	(*Tooling position to load parts*)
	Tool_At_Load.0:=
				(((Model_ID=1) OR (Model_ID>3))		(*Model 504, 526, 536, 550, 571*)
				AND Clamp1RETD AND Clamp2RETD AND Clamp3RETD AND Clamp4RETD
				AND Clamp5RETD AND Clamp6RETD AND Clamp7RETD AND Clamp8RETD
				AND Clamp9RETD AND Clamp10RETD AND Clamp11RETD AND Clamp12RETD
				AND Clamp13RETD AND Clamp14RETD AND Clamp15RETD AND Clamp16RETD
				AND Clamp17RETD AND Clamp18RETD AND Clamp19RETD AND Clamp20RETD
				AND Clamp21RETD AND Clamp22RETD AND Pin1ADVD AND Pin2ADVD AND Pin3ADVD AND Pin4ADVD 
				AND Pin5RETD AND Pin6RETD AND Pin7ADVD AND Pin8ADVD AND Pin9ADVD AND Pin10ADVD 
				AND Pin11ADVD AND Pin12ADVD AND Pin13ADVD AND Pin14RETD AND Pin15RETD AND Pin16ADVD AND Pin17ADVD 
				AND Pin18ADVD AND Slide1ADVD AND Slide2ADVD AND Slide3RETD AND Slide4RETD AND Slide5RETD AND Slide6RETD
				AND Slide7RETD AND Slide8RETD AND Slide9RETD AND Slide10ADVD AND Slide11RETD AND Slide12RETD
				AND Slide13ADVD AND Slide14ADVD AND Swing1RETD AND Swing2RETD AND Swing3RETD)
			OR
				((Model_ID=2)		(*Model 524*)
				AND Clamp1RETD AND Clamp2RETD AND Clamp3RETD AND Clamp4RETD
				AND Clamp5RETD AND Clamp6RETD AND Clamp7RETD AND Clamp8RETD
				AND Clamp9RETD AND Clamp10RETD AND Clamp11RETD AND Clamp12RETD
				AND Clamp13RETD AND Clamp14RETD AND Clamp15RETD AND Clamp16RETD
				AND Clamp17RETD AND Clamp18RETD AND Clamp19RETD AND Clamp20RETD
				AND Clamp21RETD AND Clamp22RETD AND Pin1ADVD AND Pin2ADVD AND Pin3ADVD AND Pin4ADVD 
				AND Pin5ADVD AND Pin6RETD AND Pin7ADVD AND Pin8ADVD AND Pin9ADVD AND Pin10ADVD 
				AND Pin11ADVD AND Pin12ADVD AND Pin13ADVD AND Pin14RETD AND Pin15ADVD AND Pin16ADVD AND Pin17ADVD 
				AND Pin18ADVD AND Slide1ADVD AND Slide2ADVD AND Slide3RETD AND Slide4RETD AND Slide5RETD AND Slide6RETD
				AND Slide7RETD AND Slide8RETD AND Slide9RETD AND Slide10ADVD AND Slide11RETD AND Slide12RETD
				AND Slide13ADVD AND Slide14ADVD AND Swing1RETD AND Swing2RETD AND Swing3RETD)
			OR
				((Model_ID=3)		(*Model 543*)
				AND Clamp1RETD AND Clamp2RETD AND Clamp3RETD AND Clamp4RETD
				AND Clamp5RETD AND Clamp6RETD AND Clamp7RETD AND Clamp8RETD
				AND Clamp9RETD AND Clamp10RETD AND Clamp11RETD AND Clamp12RETD
				AND Clamp13RETD AND Clamp14RETD AND Clamp15RETD AND Clamp16RETD
				AND Clamp17RETD AND Clamp18RETD AND Clamp19RETD AND Clamp20RETD
				AND Clamp21RETD AND Clamp22RETD AND Pin1ADVD AND Pin2ADVD AND Pin3ADVD AND Pin4ADVD 
				AND Pin5RETD AND Pin6ADVD AND Pin7ADVD AND Pin8ADVD AND Pin9ADVD AND Pin10ADVD 
				AND Pin11ADVD AND Pin12ADVD AND Pin13ADVD AND Pin14ADVD AND Pin15RETD AND Pin16ADVD AND Pin17ADVD 
				AND Pin18ADVD AND Slide1ADVD AND Slide2ADVD AND Slide3RETD AND Slide4RETD AND Slide5RETD AND Slide6RETD
				AND Slide7RETD AND Slide8RETD AND Slide9RETD AND Slide10ADVD AND Slide11RETD AND Slide12RETD
				AND Slide13ADVD AND Slide14ADVD AND Swing1RETD AND Swing2RETD AND Swing3RETD);
	
	(*Tooling position on Loading Complete*)	
	Tool_At_Load.1:= 
				(((Model_ID=1) OR (Model_ID>3))		(*Model 504, 526, 536, 550, 571*)
				AND Clamp1ADVD AND Clamp2ADVD AND Clamp3ADVD AND Clamp4ADVD AND Clamp5ADVD AND Clamp5ADVD AND Clamp5ADVD
				AND Clamp6ADVD AND Clamp7ADVD AND Clamp8ADVD AND Clamp9ADVD AND Clamp10ADVD AND Clamp11ADVD AND Clamp12ADVD
				AND Clamp13ADVD AND Clamp14ADVD AND Clamp15ADVD AND Clamp16ADVD AND Clamp17ADVD AND Clamp18ADVD AND Clamp19ADVD
				AND Clamp20ADVD AND Clamp21ADVD AND Clamp22ADVD AND Pin1ADVD AND Pin2ADVD AND Pin3ADVD AND Pin4ADVD AND Pin5RETD
				AND Pin6RETD AND Pin7ADVD AND Pin8ADVD AND Pin9ADVD AND Pin10ADVD AND Pin11ADVD AND Pin12ADVD AND Pin13ADVD
				AND Pin14RETD AND Pin15RETD AND Pin16ADVD AND Pin17ADVD AND Pin18ADVD AND Slide1ADVD AND Slide2ADVD AND Slide3ADVD
				AND Slide4ADVD AND Slide5ADVD AND Slide6ADVD AND Slide7ADVD AND Slide8ADVD AND Slide9ADVD AND Slide10ADVD AND Slide11ADVD
				AND Slide12ADVD AND Slide13ADVD AND Slide14ADVD AND Swing1ADVD AND Swing2ADVD AND Swing3ADVD)
			OR
				((Model_ID=2)		(*Model 524*)
				AND Clamp1ADVD AND Clamp2ADVD AND Clamp3ADVD AND Clamp4ADVD AND Clamp5ADVD AND Clamp5ADVD AND Clamp5ADVD
				AND Clamp6ADVD AND Clamp7ADVD AND Clamp8ADVD AND Clamp9ADVD AND Clamp10ADVD AND Clamp11ADVD AND Clamp12ADVD
				AND Clamp13ADVD AND Clamp14ADVD AND Clamp15ADVD AND Clamp16ADVD AND Clamp17ADVD AND Clamp18ADVD AND Clamp19ADVD
				AND Clamp20ADVD AND Clamp21ADVD AND Clamp22ADVD AND Pin1ADVD AND Pin2ADVD AND Pin3ADVD AND Pin4ADVD AND Pin5ADVD
				AND Pin6RETD AND Pin7ADVD AND Pin8ADVD AND Pin9ADVD AND Pin10ADVD AND Pin11ADVD AND Pin12ADVD AND Pin13ADVD
				AND Pin14RETD AND Pin15ADVD AND Pin16ADVD AND Pin17ADVD AND Pin18ADVD AND Slide1ADVD AND Slide2ADVD AND Slide3ADVD
				AND Slide4ADVD AND Slide5ADVD AND Slide6ADVD AND Slide7ADVD AND Slide8ADVD AND Slide9ADVD AND Slide10ADVD AND Slide11ADVD
				AND Slide12ADVD AND Slide13ADVD AND Slide14ADVD AND Swing1ADVD AND Swing2ADVD AND Swing3ADVD)
			OR
				((Model_ID=3)		(*Model 543*)
				AND Clamp1ADVD AND Clamp2ADVD AND Clamp3ADVD AND Clamp4ADVD AND Clamp5ADVD AND Clamp5ADVD AND Clamp5ADVD
				AND Clamp6ADVD AND Clamp7ADVD AND Clamp8ADVD AND Clamp9ADVD AND Clamp10ADVD AND Clamp11ADVD AND Clamp12ADVD
				AND Clamp13ADVD AND Clamp14ADVD AND Clamp15ADVD AND Clamp16ADVD AND Clamp17ADVD AND Clamp18ADVD AND Clamp19ADVD
				AND Clamp20ADVD AND Clamp21ADVD AND Clamp22ADVD AND Pin1ADVD AND Pin2ADVD AND Pin3ADVD AND Pin4ADVD AND Pin5RETD
				AND Pin6ADVD AND Pin7ADVD AND Pin8ADVD AND Pin9ADVD AND Pin10ADVD AND Pin11ADVD AND Pin12ADVD AND Pin13ADVD
				AND Pin14ADVD AND Pin15RETD AND Pin16ADVD AND Pin17ADVD AND Pin18ADVD AND Slide1ADVD AND Slide2ADVD AND Slide3ADVD
				AND Slide4ADVD AND Slide5ADVD AND Slide6ADVD AND Slide7ADVD AND Slide8ADVD AND Slide9ADVD AND Slide10ADVD AND Slide11ADVD
				AND Slide12ADVD AND Slide13ADVD AND Slide14ADVD AND Swing1ADVD AND Swing2ADVD AND Swing3ADVD);
	(*Tool Position for Calling in Load Robots*)
	Tool_At_Load.2:=  
				(((Model_ID=1) OR (Model_ID>3))		(*Model 504, 526, 536, 550, 571*)
				AND Clamp1ADVD AND Clamp2ADVD AND Clamp3ADVD AND Clamp4ADVD AND Clamp5ADVD
				AND Clamp6RETD AND Clamp7RETD AND Clamp8RETD AND Clamp9ADVD AND Clamp10ADVD AND Clamp11RETD AND Clamp12ADVD
				AND Clamp13ADVD AND Clamp14ADVD AND Clamp15RETD AND Clamp16ADVD AND Clamp17RETD AND Clamp18ADVD AND Clamp19RETD
				AND Clamp20RETD AND Clamp21ADVD AND Clamp22ADVD AND Pin1ADVD AND Pin2ADVD AND Pin3ADVD AND Pin4ADVD AND Pin5RETD
				AND Pin6RETD AND Pin7ADVD AND Pin8ADVD AND Pin9ADVD AND Pin10ADVD AND Pin11ADVD AND Pin12ADVD AND Pin13ADVD
				AND Pin14RETD AND Pin15RETD AND Pin16ADVD AND Pin17ADVD AND Pin18ADVD AND Slide1ADVD AND Slide2ADVD AND Slide3RETD
				AND Slide4RETD AND Slide5RETD AND Slide6RETD AND Slide7RETD AND Slide8RETD AND Slide9RETD AND Slide10ADVD AND Slide11RETD
				AND Slide12RETD AND Slide13ADVD AND Slide14ADVD AND Swing1RETD AND Swing2RETD AND Swing3RETD)
			OR
				((Model_ID=2)		(*Model 524*)
				AND Clamp1ADVD AND Clamp2ADVD AND Clamp3ADVD AND Clamp4ADVD AND Clamp5ADVD
				AND Clamp6ADVD AND Clamp7RETD AND Clamp8RETD AND Clamp9ADVD AND Clamp10ADVD AND Clamp11RETD AND Clamp12ADVD
				AND Clamp13ADVD AND Clamp14ADVD AND Clamp15RETD AND Clamp16ADVD AND Clamp17RETD AND Clamp18ADVD AND Clamp19RETD
				AND Clamp20ADVD AND Clamp21ADVD AND Clamp22ADVD AND Pin1ADVD AND Pin2ADVD AND Pin3ADVD AND Pin4ADVD AND Pin5ADVD
				AND Pin6RETD AND Pin7ADVD AND Pin8ADVD AND Pin9ADVD AND Pin10ADVD AND Pin11ADVD AND Pin12ADVD AND Pin13ADVD
				AND Pin14RETD AND Pin15ADVD AND Pin16ADVD AND Pin17ADVD AND Pin18ADVD AND Slide1ADVD AND Slide2ADVD AND Slide3RETD
				AND Slide4RETD AND Slide5RETD AND Slide6RETD AND Slide7RETD AND Slide8RETD AND Slide9RETD AND Slide10ADVD AND Slide11RETD
				AND Slide12RETD AND Slide13ADVD AND Slide14ADVD AND Swing1RETD AND Swing2RETD AND Swing3RETD)
			OR
				((Model_ID=3)		(*Model 543*)
				AND Clamp1ADVD AND Clamp2ADVD AND Clamp3ADVD AND Clamp4ADVD AND Clamp5ADVD
				AND Clamp6RETD AND Clamp7RETD AND Clamp8ADVD AND Clamp9ADVD AND Clamp10ADVD AND Clamp11RETD AND Clamp12ADVD
				AND Clamp13ADVD AND Clamp14ADVD AND Clamp15RETD AND Clamp16ADVD AND Clamp17RETD AND Clamp18ADVD AND Clamp19ADVD
				AND Clamp20RETD AND Clamp21ADVD AND Clamp22ADVD AND Pin1ADVD AND Pin2ADVD AND Pin3ADVD AND Pin4ADVD AND Pin5RETD
				AND Pin6ADVD AND Pin7ADVD AND Pin8ADVD AND Pin9ADVD AND Pin10ADVD AND Pin11ADVD AND Pin12ADVD AND Pin13ADVD
				AND Pin14ADVD AND Pin15RETD AND Pin16ADVD AND Pin17ADVD AND Pin18ADVD AND Slide1ADVD AND Slide2ADVD AND Slide3RETD
				AND Slide4RETD AND Slide5RETD AND Slide6RETD AND Slide7RETD AND Slide8RETD AND Slide9RETD AND Slide10ADVD AND Slide11RETD
				AND Slide12RETD AND Slide13ADVD AND Slide14ADVD AND Swing1RETD AND Swing2RETD AND Swing3RETD);
	Tool_At_Load.3:= FALSE;
	Tool_At_Load.4:= FALSE;


	Tool_At_Seal.0:= FALSE;
	Tool_At_Seal.1:= FALSE;
	Tool_At_Seal.2:= FALSE;
	Tool_At_Seal.3:= FALSE;
	Tool_At_Seal.4:= FALSE;


	Tool_At_Stud.0:= FALSE;
	Tool_At_Stud.1:= FALSE;
	Tool_At_Stud.2:= FALSE;
	Tool_At_Stud.3:= FALSE;
	Tool_At_Stud.4:= FALSE;

	(*Tooling position for ready to rotate*)
	Tool_At_Rotate.0:= 
				(((Model_ID=1) OR (Model_ID>3))		(*Model 504, 526, 536, 550, 571*)
				AND Clamp1ADVD AND Clamp2ADVD AND Clamp3ADVD AND Clamp4ADVD AND Clamp5ADVD
				AND Clamp6RETD AND Clamp7RETD AND Clamp8RETD AND Clamp9ADVD AND Clamp10ADVD AND Clamp11RETD AND Clamp12ADVD
				AND Clamp13ADVD AND Clamp14ADVD AND Clamp15RETD AND Clamp16ADVD AND Clamp17RETD AND Clamp18ADVD AND Clamp19RETD
				AND Clamp20RETD AND Clamp21ADVD AND Clamp22ADVD AND Pin1ADVD AND Pin2ADVD AND Pin3ADVD AND Pin4ADVD AND Pin5RETD
				AND Pin6RETD AND Pin7ADVD AND Pin8ADVD AND Pin9ADVD AND Pin10ADVD AND Pin11ADVD AND Pin12ADVD AND Pin13ADVD
				AND Pin14RETD AND Pin15RETD AND Pin16ADVD AND Pin17ADVD AND Pin18ADVD AND Slide1ADVD AND Slide2ADVD AND Slide3RETD
				AND Slide4RETD AND Slide5RETD AND Slide6RETD AND Slide7RETD AND Slide8RETD AND Slide9RETD AND Slide10ADVD AND Slide11RETD
				AND Slide12RETD AND Slide13ADVD AND Slide14ADVD AND Swing1RETD AND Swing2RETD AND Swing3RETD)
			OR
				((Model_ID=2)		(*Model 524*)
				AND Clamp1ADVD AND Clamp2ADVD AND Clamp3ADVD AND Clamp4ADVD AND Clamp5ADVD
				AND Clamp6ADVD AND Clamp7RETD AND Clamp8RETD AND Clamp9ADVD AND Clamp10ADVD AND Clamp11RETD AND Clamp12ADVD
				AND Clamp13ADVD AND Clamp14ADVD AND Clamp15RETD AND Clamp16ADVD AND Clamp17RETD AND Clamp18ADVD AND Clamp19RETD
				AND Clamp20ADVD AND Clamp21ADVD AND Clamp22ADVD AND Pin1ADVD AND Pin2ADVD AND Pin3ADVD AND Pin4ADVD AND Pin5ADVD
				AND Pin6RETD AND Pin7ADVD AND Pin8ADVD AND Pin9ADVD AND Pin10ADVD AND Pin11ADVD AND Pin12ADVD AND Pin13ADVD
				AND Pin14RETD AND Pin15ADVD AND Pin16ADVD AND Pin17ADVD AND Pin18ADVD AND Slide1ADVD AND Slide2ADVD AND Slide3RETD
				AND Slide4RETD AND Slide5RETD AND Slide6RETD AND Slide7RETD AND Slide8RETD AND Slide9RETD AND Slide10ADVD AND Slide11RETD
				AND Slide12RETD AND Slide13ADVD AND Slide14ADVD AND Swing1RETD AND Swing2RETD AND Swing3RETD)
			OR
				((Model_ID=3)		(*Model 543*)
				AND Clamp1ADVD AND Clamp2ADVD AND Clamp3ADVD AND Clamp4ADVD AND Clamp5ADVD
				AND Clamp6RETD AND Clamp7RETD AND Clamp8ADVD AND Clamp9ADVD AND Clamp10ADVD AND Clamp11RETD AND Clamp12ADVD
				AND Clamp13ADVD AND Clamp14ADVD AND Clamp15RETD AND Clamp16ADVD AND Clamp17RETD AND Clamp18ADVD AND Clamp19ADVD
				AND Clamp20RETD AND Clamp21ADVD AND Clamp22ADVD AND Pin1ADVD AND Pin2ADVD AND Pin3ADVD AND Pin4ADVD AND Pin5RETD
				AND Pin6ADVD AND Pin7ADVD AND Pin8ADVD AND Pin9ADVD AND Pin10ADVD AND Pin11ADVD AND Pin12ADVD AND Pin13ADVD
				AND Pin14ADVD AND Pin15RETD AND Pin16ADVD AND Pin17ADVD AND Pin18ADVD AND Slide1ADVD AND Slide2ADVD AND Slide3RETD
				AND Slide4RETD AND Slide5RETD AND Slide6RETD AND Slide7RETD AND Slide8RETD AND Slide9RETD AND Slide10ADVD AND Slide11RETD
				AND Slide12RETD AND Slide13ADVD AND Slide14ADVD AND Swing1RETD AND Swing2RETD AND Swing3RETD);
				
	Tool_At_Rotate.1:= FALSE;
	Tool_At_Rotate.2:= FALSE;
	Tool_At_Rotate.3:= FALSE;
	Tool_At_Rotate.4:= FALSE;

	(*Tooling position for welding*)
	Tool_At_Weld.0:= 
				(((Model_ID=1) OR (Model_ID>3))		(*Model 504, 526, 536, 550, 571*)
				AND Clamp1ADVD AND Clamp2ADVD AND Clamp3ADVD AND Clamp4ADVD AND Clamp5ADVD AND Clamp5ADVD AND Clamp5ADVD
				AND Clamp6RETD AND Clamp7ADVD AND Clamp8RETD AND Clamp9ADVD AND Clamp10ADVD AND Clamp11ADVD AND Clamp12ADVD
				AND Clamp13ADVD AND Clamp14ADVD AND Clamp15ADVD AND Clamp16ADVD AND Clamp17ADVD AND Clamp18ADVD AND Clamp19RETD
				AND Clamp20RETD AND Clamp21ADVD AND Clamp22ADVD AND Pin1ADVD AND Pin2ADVD AND Pin3ADVD AND Pin4ADVD AND Pin5RETD
				AND Pin6RETD AND Pin7ADVD AND Pin8ADVD AND Pin9ADVD AND Pin10ADVD AND Pin11ADVD AND Pin12ADVD AND Pin13ADVD
				AND Pin14RETD AND Pin15RETD AND Pin16ADVD AND Pin17ADVD AND Pin18ADVD AND Slide1ADVD AND Slide2ADVD AND Slide3ADVD
				AND Slide4RETD AND Slide5ADVD AND Slide6ADVD AND Slide7ADVD AND Slide8ADVD AND Slide9ADVD AND Slide10ADVD AND Slide11RETD
				AND Slide12ADVD AND Slide13ADVD AND Slide14ADVD AND Swing1RETD AND Swing2ADVD AND Swing3RETD)
			OR
				((Model_ID=2)		(*Model 524*)
				AND Clamp1ADVD AND Clamp2ADVD AND Clamp3ADVD AND Clamp4ADVD AND Clamp5ADVD AND Clamp5ADVD AND Clamp5ADVD
				AND Clamp6ADVD AND Clamp7ADVD AND Clamp8RETD AND Clamp9ADVD AND Clamp10ADVD AND Clamp11ADVD AND Clamp12ADVD
				AND Clamp13ADVD AND Clamp14ADVD AND Clamp15ADVD AND Clamp16ADVD AND Clamp17ADVD AND Clamp18ADVD AND Clamp19RETD
				AND Clamp20ADVD AND Clamp21ADVD AND Clamp22ADVD AND Pin1ADVD AND Pin2ADVD AND Pin3ADVD AND Pin4ADVD AND Pin5ADVD
				AND Pin6RETD AND Pin7ADVD AND Pin8ADVD AND Pin9ADVD AND Pin10ADVD AND Pin11ADVD AND Pin12ADVD AND Pin13ADVD
				AND Pin14RETD AND Pin15ADVD AND Pin16ADVD AND Pin17ADVD AND Pin18ADVD AND Slide1ADVD AND Slide2ADVD AND Slide3ADVD
				AND Slide4ADVD AND Slide5ADVD AND Slide6ADVD AND Slide7ADVD AND Slide8ADVD AND Slide9ADVD AND Slide10ADVD AND Slide11ADVD
				AND Slide12ADVD AND Slide13ADVD AND Slide14ADVD AND Swing1RETD AND Swing2ADVD AND Swing3RETD)
			OR
				((Model_ID=3)		(*Model 543*)
				AND Clamp1ADVD AND Clamp2ADVD AND Clamp3ADVD AND Clamp4ADVD AND Clamp5ADVD AND Clamp5ADVD AND Clamp5ADVD
				AND Clamp6RETD AND Clamp7ADVD AND Clamp8ADVD AND Clamp9ADVD AND Clamp10ADVD AND Clamp11ADVD AND Clamp12ADVD
				AND Clamp13ADVD AND Clamp14ADVD AND Clamp15ADVD AND Clamp16ADVD AND Clamp17ADVD AND Clamp18ADVD AND Clamp19ADVD
				AND Clamp20RETD AND Clamp21ADVD AND Clamp22ADVD AND Pin1ADVD AND Pin2ADVD AND Pin3ADVD AND Pin4ADVD AND Pin5RETD
				AND Pin6ADVD AND Pin7ADVD AND Pin8ADVD AND Pin9ADVD AND Pin10ADVD AND Pin11ADVD AND Pin12ADVD AND Pin13ADVD
				AND Pin14ADVD AND Pin15RETD AND Pin16ADVD AND Pin17ADVD AND Pin18ADVD AND Slide1ADVD AND Slide2ADVD AND Slide3ADVD
				AND Slide4RETD AND Slide5ADVD AND Slide6ADVD AND Slide7ADVD AND Slide8ADVD AND Slide9ADVD AND Slide10ADVD AND Slide11RETD
				AND Slide12ADVD AND Slide13ADVD AND Slide14ADVD AND Swing1ADVD AND Swing2ADVD AND Swing3ADVD);
	Tool_At_Weld.1:= FALSE;
	Tool_At_Weld.2:= FALSE;
	Tool_At_Weld.3:= FALSE;
	Tool_At_Weld.4:= FALSE;

	(*Tooling position for unload*)
	Tool_At_Unload.0:=Clamp1RETD AND Clamp2RETD AND Clamp3RETD AND Clamp4RETD
				AND Clamp5RETD AND Clamp6RETD AND Clamp7ADVD AND Clamp8RETD
				AND Clamp9RETD AND Clamp10RETD AND Clamp11ADVD AND Clamp12RETD
				AND Clamp13RETD AND Clamp14RETD AND Clamp15ADVD AND Clamp16RETD
				AND Clamp17ADVD AND Clamp18RETD AND Clamp19RETD AND Clamp20RETD
				AND Clamp21RETD AND Clamp22RETD AND Pin1RETD AND Pin2RETD AND Pin3RETD AND Pin4RETD AND Pin5RETD
				AND Pin6RETD AND Pin7RETD AND Pin8RETD AND Pin9RETD AND Pin10RETD AND Pin11RETD AND Pin12RETD 
				AND Pin13RETD AND Pin14RETD AND Pin15RETD AND Pin16RETD AND Pin17RETD AND Pin18RETD
				AND Slide1RETD AND Slide2RETD AND Slide3RETD AND Slide4RETD AND Slide5RETD AND Slide6RETD
				AND Slide7RETD AND Slide8RETD AND Slide9RETD AND Slide10RETD AND Slide11RETD AND Slide12RETD
				AND Slide13RETD AND Slide14RETD AND Swing1RETD AND Swing2RETD AND Swing3RETD;
	
	Tool_At_Unload.1:=Clamp1RETD AND Clamp2RETD AND Clamp3RETD AND Clamp4RETD
				AND Clamp5RETD AND Clamp6RETD AND Clamp7RETD AND Clamp8RETD
				AND Clamp9RETD AND Clamp10RETD AND Clamp11RETD AND Clamp12RETD
				AND Clamp13RETD AND Clamp14RETD AND Clamp15RETD AND Clamp16RETD
				AND Clamp17RETD AND Clamp18RETD AND Clamp19RETD AND Clamp20RETD
				AND Clamp21RETD AND Clamp22RETD AND Pin1RETD AND Pin2RETD AND Pin3RETD AND Pin4RETD AND Pin5RETD
				AND Pin6RETD AND Pin7RETD AND Pin8RETD AND Pin9RETD AND Pin10RETD AND Pin11RETD AND Pin12RETD 
				AND Pin13RETD AND Pin14RETD AND Pin15RETD AND Pin16RETD AND Pin17RETD AND Pin18RETD
				AND Slide1RETD AND Slide2RETD AND Slide3RETD AND Slide4RETD AND Slide5RETD AND Slide6RETD
				AND Slide7RETD AND Slide8RETD AND Slide9RETD AND Slide10RETD AND Slide11RETD AND Slide12RETD
				AND Slide13RETD AND Slide14RETD AND Swing1RETD AND Swing2RETD AND Swing3RETD;
	Tool_At_Unload.2:= FALSE;
	Tool_At_Unload.3:= FALSE;
	Tool_At_Unload.4:= FALSE;







































(*end*)
END_ACTION

ACTION Tool_VBSeq_Repos:
(*+++++++++++THIS AREA IS CUSTOM PER INSTALLATION AND WILL HAVE TO BE MODIFIED PER +++++++++++++*)
(*+++++++++++THIS AREA IS CUSTOM PER INSTALLATION AND WILL HAVE TO BE MODIFIED PER +++++++++++++*)


(*!!!!!!!!!!!!!!!!!!!!!!!!!!!!!!!!!!!!!!!!!! Tool Motion Control !!!!!!!!!!!!!!!!!!!!!!!!!!!!!!!*)

(*----------------------------------------- Clamp / Unclamp Steps -------------------------------*)

(*$$$$$$$$$$$$$$$$$$$$$$$$$$$$$$$$$$ Develop Clamp and Unclamp Interlocks $$$$$$$$$$$$$$$$$$$$$$*)
(* Note: This is one method to create valve bank commands for clamp and unclamp sequencing
you are welcome to use the direct method as well*)


	(*---------------------------------------------------------Start Clamp Sequence---------------------------------------------------------*)
	
	(*First Stage Clamping*)		(*V8, V10 ADV, IF Model 2 then V2 ADV, IF Model 3 then V5 ADV*)
	Clamp_Step.0:= Auto_Run AND NOT Welding_Complete OR (Cycle_Complete AND NOT Tool_At_Home AND All_Sensors_Off);
	
	
	(*Second Stage Clamping*)		(*V7, V9, V11 ADV, IF Model 2 then V1 ADV, IF Model 3 V4 ADV*)
	
	(*Model 504, 526, 536, 550, 571*)
	IF (Model_ID=1) OR (Model_ID>3) THEN		
				Clamp_Step.1:=  Clamp_Step.0 AND (Load_Complete1 OR Load_Complete2) AND
								(*V8*)
								(Pin1ADVD AND Pin2ADVD AND Pin3ADVD AND Pin4ADVD AND Pin7ADVD 
								AND Pin9ADVD AND Pin16ADVD AND Pin17ADVD AND Pin18ADVD AND Slide10ADVD)
								(*V10*)
								AND (Pin8ADVD AND Pin10ADVD AND Pin11ADVD AND Pin12ADVD AND Pin13ADVD 
								AND Slide1ADVD AND Slide2ADVD AND Slide13ADVD AND Slide14ADVD);
		(*Model 524*)						
		ELSIF (Model_ID=2) THEN					
				Clamp_Step.1:=  Clamp_Step.0 AND (Load_Complete1 OR Load_Complete2) AND
								(*V2*)
								(Pin5ADVD AND Pin15ADVD)
								(*V8*)
								AND (Pin1ADVD AND Pin2ADVD AND Pin3ADVD AND Pin4ADVD AND Pin7ADVD 
								AND Pin9ADVD AND Pin16ADVD AND Pin17ADVD AND Pin18ADVD AND Slide10ADVD)
								(*V10*)
								AND (Pin8ADVD AND Pin10ADVD AND Pin11ADVD AND Pin12ADVD AND Pin13ADVD 
								AND Slide1ADVD AND Slide2ADVD AND Slide13ADVD AND Slide14ADVD);
		(*Model 543*)			
		ELSIF (Model_ID=3) THEN					
				Clamp_Step.1:=  Clamp_Step.0 AND (Load_Complete1 OR Load_Complete2) AND 
								(*V5*)
								(Pin6ADVD AND Pin14ADVD)
								(*V8*)
								AND (Pin1ADVD AND Pin2ADVD AND Pin3ADVD AND Pin4ADVD AND Pin7ADVD 
								AND Pin9ADVD AND Pin16ADVD AND Pin17ADVD AND Pin18ADVD AND Slide10ADVD)
								(*V10*)
								AND (Pin8ADVD AND Pin10ADVD AND Pin11ADVD AND Pin12ADVD AND Pin13ADVD 
								AND Slide1ADVD AND Slide2ADVD AND Slide13ADVD AND Slide14ADVD);						
	END_IF

	
	(*Third Stage Clamping*)		(*V13 ADV*)
	
	(*Model 504, 526, 536, 550, 571*)
	IF (Model_ID=1) OR (Model_ID>3) THEN
				Clamp_Step.2:= 	Clamp_Step.1 AND (All_Sensors_On.2 OR Clamp_Step.2) AND Repo_Reqs.0 AND
								(*V7*)
								(Clamp3ADVD AND Clamp18ADVD)
								(*V9*)
								AND (Clamp1ADVD AND Clamp2ADVD AND Clamp4ADVD AND Clamp5ADVD AND Clamp10ADVD 
								AND Clamp14ADVD AND Clamp21ADVD AND Clamp22ADVD)
								(*V11*)
								AND (Clamp9ADVD AND Clamp12ADVD AND Clamp13ADVD AND Clamp16ADVD);

		ELSIF (Model_ID=2) THEN
				Clamp_Step.2:= 	Clamp_Step.1 AND (All_Sensors_On.2 OR Clamp_Step.2) AND Repo_Reqs.0 AND
								(*V7*)
								(Clamp3ADVD AND Clamp18ADVD)
								(*V9*)
								AND (Clamp1ADVD AND Clamp2ADVD AND Clamp4ADVD AND Clamp5ADVD AND Clamp10ADVD 
								AND Clamp14ADVD AND Clamp21ADVD AND Clamp22ADVD)
								(*V11*)
								AND (Clamp9ADVD AND Clamp12ADVD AND Clamp13ADVD AND Clamp16ADVD)
								(*V1*)
								AND (Clamp6ADVD AND Clamp20ADVD);
		ELSIF (Model_ID=3) THEN
				Clamp_Step.2:= 	Clamp_Step.1 AND (All_Sensors_On.2 OR Clamp_Step.2) AND Repo_Reqs.0 AND
								(*V7*)
								(Clamp3ADVD AND Clamp18ADVD)
								(*V9*)
								AND (Clamp1ADVD AND Clamp2ADVD AND Clamp4ADVD AND Clamp5ADVD AND Clamp10ADVD 
								AND Clamp14ADVD AND Clamp21ADVD AND Clamp22ADVD)
								(*V11*)
								AND (Clamp9ADVD AND Clamp12ADVD AND Clamp13ADVD AND Clamp16ADVD)
								(*V4*)
								AND (Clamp8ADVD AND Clamp19ADVD);
	END_IF


	(*Forth Stage Clamping*)		(*V12 ADV, IF Model 2 V3 ADV, IF Model 3 V6 ADV*)
	
	Clamp_Step.3:= Clamp_Step.2 AND Repo_Reqs.0 AND
					(*V13*)
					(Clamp7ADVD AND Clamp11ADVD AND Clamp15ADVD AND Clamp17ADVD);




	(*---------------------------------------------------------Start Unclamp Sequence---------------------------------------------------------*)

	(*First Stage Unclamping*)		(*V7, V9, V11 RET, IF Model 2 V1 RET, IF Model 3 V4 RET*)

	Unclamp_Step.0:= (Welding_Complete AND TurnTableA_At_Robot);


	(*Second Stage Unclamping*)		(*V8, V10 RET, IF Model 2 V2 RET, IF Model 3 V5 RET*)
	(*Model 504, 526, 536, 550, 571*)
	IF (Model_ID=1) OR (Model_ID>3) THEN
			Unclamp_Step.1:= Unclamp_Step.0 AND 
								(*V7*)
								(Clamp3RETD AND Clamp18RETD)
								(*V9*)
								AND (Clamp1RETD AND Clamp2RETD AND Clamp4RETD AND Clamp5RETD AND Clamp10RETD AND Clamp14RETD AND Clamp21RETD AND Clamp22RETD)
								(*V11*)
								AND (Clamp9RETD AND Clamp12RETD AND Clamp13RETD AND Clamp16RETD);
		(*Model 524*)							
		ELSIF (Model_ID=2) THEN
				Unclamp_Step.1:= Unclamp_Step.0 AND 
									(*V7*)
									(Clamp3RETD AND Clamp18RETD)
									(*V9*)
									AND (Clamp1RETD AND Clamp2RETD AND Clamp4RETD AND Clamp5RETD AND Clamp10RETD AND Clamp14RETD AND Clamp21RETD AND Clamp22RETD)
									(*V11*)
									AND (Clamp9RETD AND Clamp12RETD AND Clamp13RETD AND Clamp16RETD)
									(*V1*)
									AND (Clamp6RETD AND Clamp20RETD);
		(*Model 543*)
		ELSIF (Model_ID=3) THEN							
				Unclamp_Step.1:= Unclamp_Step.0 AND 
									(*V7*)
									(Clamp3RETD AND Clamp18RETD)
									(*V9*)
									AND (Clamp1RETD AND Clamp2RETD AND Clamp4RETD AND Clamp5RETD AND Clamp10RETD AND Clamp14RETD AND Clamp21RETD AND Clamp22RETD)
									(*V11*)
									AND (Clamp9RETD AND Clamp12RETD AND Clamp13RETD AND Clamp16RETD)
									(*V4*)
									AND (Clamp8RETD AND Clamp19RETD);
	END_IF

	
	(*Third Stage Unclamping*)		(*V12 RET, IF Model 2 V3 RET, IF Model 3 V6 RET*)
	(*Model 504, 526, 536, 550, 571*)
	IF (Model_ID=1) OR (Model_ID>3) THEN
			Unclamp_Step.2:= Unclamp_Step.1 AND 
						(*V8*)
						(Pin1RETD AND Pin2RETD AND Pin3RETD AND Pin4RETD AND Pin7RETD AND Pin9RETD AND Pin16RETD AND Pin17RETD AND Pin18RETD AND Slide10RETD)
						(*V10*)
						AND (Pin8RETD AND Pin10RETD AND Pin11RETD AND Pin12RETD AND Pin13RETD AND Slide1RETD AND Slide2RETD AND Slide13RETD AND Slide14RETD);
		(*Model 524*)
		ELSIF (Model_ID=2) THEN
				Unclamp_Step.2:= Unclamp_Step.1 AND 
							(*V8*)
							(Pin1RETD AND Pin2RETD AND Pin3RETD AND Pin4RETD AND Pin7RETD AND Pin9RETD AND Pin16RETD AND Pin17RETD AND Pin18RETD AND Slide10RETD)
							(*V10*)
							AND (Pin8RETD AND Pin10RETD AND Pin11RETD AND Pin12RETD AND Pin13RETD AND Slide1RETD AND Slide2RETD AND Slide13RETD AND Slide14RETD)
							(*V2*)
							AND (Pin5RETD AND Pin15RETD);
		(*Model 543*)
		ELSIF (Model_ID=3) THEN
				Unclamp_Step.2:= Unclamp_Step.1 AND 
							(*V8*)
							(Pin1RETD AND Pin2RETD AND Pin3RETD AND Pin4RETD AND Pin7RETD AND Pin9RETD AND Pin16RETD AND Pin17RETD AND Pin18RETD AND Slide10RETD)
							(*V10*)
							AND (Pin8RETD AND Pin10RETD AND Pin11RETD AND Pin12RETD AND Pin13RETD AND Slide1RETD AND Slide2RETD AND Slide13RETD AND Slide14RETD)
							(*V5*)
							AND (Pin6RETD AND Pin14RETD);
	
	END_IF

	(*Fourth Stage Unclamping*)		(*V13 RET*)
	(*Model 504, 526, 536, 550, 571*)
	IF (Model_ID=1) OR (Model_ID>3) THEN
				Unclamp_Step.3:= Unclamp_Step.2 AND Repo_Reqs.1 AND
							(*V12*)
							(Slide3RETD AND Slide5RETD AND Slide6RETD AND Slide7RETD AND Slide8RETD AND Slide9RETD AND Slide12RETD AND Swing2RETD);

		ELSIF (Model_ID=2) THEN
				Unclamp_Step.3:= Unclamp_Step.2 AND Repo_Reqs.1 AND 
							(*V12*)
							(Slide3RETD AND Slide5RETD AND Slide6RETD AND Slide7RETD AND Slide8RETD AND Slide9RETD AND Slide12RETD AND Swing2RETD)
							(*V3*)
							AND (Slide4RETD AND Slide11RETD);
							
							
		ELSIF (Model_ID=3) THEN
				Unclamp_Step.3:= Unclamp_Step.2 AND Repo_Reqs.1 AND 
							(*V12*)
							(Slide3RETD AND Slide5RETD AND Slide6RETD AND Slide7RETD AND Slide8RETD AND Slide9RETD AND Slide12RETD AND Swing2RETD)
							(*V6*)
							AND (Swing1RETD AND Swing3RETD);
							
	END_IF							


(*------------------------------------------- Repositions --------------------------------------*)

	(*Reposition Request#1*)
	IF (MAIN.R4.Peripheral_Req.0 AND (MAIN.R4.Task_ID_Ack=DropOff_Fix03))
		THEN
			Repo_Reqs.0:= TRUE;
	END_IF;

	(*Reposition Request#2*)
	IF (MAIN.R4.Peripheral_Req.1 AND (MAIN.R4.Task_ID_Ack=Pickup_Fix03))
		THEN
			Repo_Reqs.1:= TRUE;
	END_IF;

	(*Reposition Request#3*)
	IF FALSE
		THEN
			Repo_Reqs.2:= TRUE;
	END_IF;

	(*Reposition Request#4*)
	IF FALSE
		THEN
			Repo_Reqs.3:= TRUE;
	END_IF;

	(*Reposition Request#5*)
	IF FALSE
		THEN
			Repo_Reqs.4:= TRUE;
	END_IF;

	(*Reposition Request#6*)
	IF FALSE
		THEN
			Repo_Reqs.5:= TRUE;
	END_IF;

	(*Reposition Request#7*)
	IF FALSE
		THEN
			Repo_Reqs.6:= TRUE;
	END_IF;

	(*Reposition Request#8*)
	IF FALSE
		THEN
			Repo_Reqs.7:= TRUE;
	END_IF;

	(*Reset All Reposition Acks At the End Of Cycle*)
	IF Cycle_Complete
		THEN
			Repo_Reqs:= 0;
	END_IF;

(*------------------------- Reposition Acks ---------------------*)
	Repo_Ack.0:= Repo_Reqs.0 AND All_Sensors_On.2 AND Tool_At_Weld.0;
	Repo_Ack.1:= Repo_Reqs.1 AND All_Sensors_On.8 AND Tool_At_Unload.1;
	Repo_Ack.2:= Repo_Reqs.2 AND FALSE;
	Repo_Ack.3:= Repo_Reqs.3 AND FALSE;
	Repo_Ack.4:= Repo_Reqs.4 AND FALSE;
	Repo_Ack.5:= Repo_Reqs.5 AND FALSE;
	Repo_Ack.6:= Repo_Reqs.6 AND FALSE;
	Repo_Ack.7:= Repo_Reqs.7 AND FALSE;
END_ACTION

ACTION ValveBank1:


(*+++++++++++THIS AREA IS CUSTOM PER INSTALLATION AND WILL HAVE TO BE MODIFIED PER +++++++++++++*)
(*+++++++++++THIS AREA IS CUSTOM PER INSTALLATION AND WILL HAVE TO BE MODIFIED PER +++++++++++++*)
(*+++++++++++THIS AREA IS CUSTOM PER INSTALLATION AND WILL HAVE TO BE MODIFIED PER +++++++++++++*)

(*+++++++++++VALVE BANK 1 +++++++++++++*)
(*+++++++++++VALVE BANK 1 +++++++++++++*)
(*+++++++++++VALVE BANK 1 +++++++++++++*)


	(*Valve 1, Model 524 ONLY*)
	(*Clamp #6, 20*)
		Valve1FB
			(
			Enable_Motion:= Enable_Motion,
			Enable_Latch:= TRUE,					(*Enabling Runs Valve as detent type (maintained solenoids*)
			Enable_SideA_PreCharge:= FALSE,		(*Enabling Turns Side A PreCharge Active, reset when Side B is energized in Auto*)
			Enable_SideB_PreCharge:= FALSE,		(*Enabling Turns Side B PreCharge Active, reset when Side A is energized in Auto*)
			PreCharge_Time:= T#0.1S,
			Enable_Auto_Commands:= In_Auto,
			Enable_Manual_Commands:= In_Manual AND (All_Robots_Clear OR TurntableB_At_Robot),  (*TLK ADDED OR*)
			In_Manual_SideA_Command:= Discrete_In.ManReqs.0,
			In_Manual_SideB_Command:= (Discrete_In.ManReqs.1 OR Discrete_In.Go_Home),
			SideA_Indicator:= (Clamp6ADVD AND Clamp20ADVD),
			SideB_Indicator:= (Clamp6RETD AND Clamp20RETD) OR Manual_Ind_HomePrompt,
			TurnOn_SideA_SOL=> N100.Q.0,
			TurnOn_SideB_SOL=> N100.Q.1,
			TurnOn_SideA_Indicator=> Manual_Indicators1.0,
			TurnOn_SideB_Indicator=> Manual_Indicators1.1
			 );
	IF (Model_ID=2) THEN		 
			Valve1FB.In_Auto_SideA_Command:= Clamp_Step.1 AND NOT Unclamp_Step.0;
			Valve1FB.In_Auto_SideB_Command:= Unclamp_Step.0 
										OR ((TurntableA_At_Robot OR Turntable_Bypassed) AND All_Sensors_Off AND Weld_Robots_Clear);
		ELSE
			Valve1FB.In_Auto_SideA_Command:= FALSE;
			Valve1FB.In_Auto_SideB_Command:= TRUE;
		END_IF

	(*Valve 2, Model 524 ONLY*)
	(*Pin #5, 15*)
		Valve2FB
			(
			Enable_Motion:= Enable_Motion,
			Enable_Latch:= TRUE,					(*Enabling Runs Valve as detent type (maintained solenoids*)
			Enable_SideA_PreCharge:= FALSE,		(*Enabling Turns Side A PreCharge Active, reset when Side B is energized in Auto*)
			Enable_SideB_PreCharge:= FALSE,		(*Enabling Turns Side B PreCharge Active, reset when Side A is energized in Auto*)
			PreCharge_Time:= T#0.10S,
			Enable_Auto_Commands:= In_Auto,
			Enable_Manual_Commands:= In_Manual AND (All_Robots_Clear OR TurntableB_At_Robot),  (*TLK ADDED OR*)
			In_Manual_SideA_Command:=  (Discrete_In.ManReqs.2 OR (Discrete_In.Go_Home AND (Model_ID = 2))),
			In_Manual_SideB_Command:= (Discrete_In.ManReqs.3 OR (Discrete_In.Go_Home AND (Model_ID <> 2))),
			SideA_Indicator:=  Pin5ADVD AND Pin15ADVD,
			SideB_Indicator:= (Pin5RETD AND Pin15RETD) OR Manual_Ind_HomePrompt,
			TurnOn_SideA_SOL=> N100.Q.2,
			TurnOn_SideB_SOL=> N100.Q.3,
			TurnOn_SideA_Indicator=> Manual_Indicators1.2,
			TurnOn_SideB_Indicator=> Manual_Indicators1.3
			 );
	IF (Model_ID=2) THEN		 
			Valve2FB.In_Auto_SideA_Command:= Clamp_Step.0 AND NOT Unclamp_Step.1
										OR ((TurntableA_At_Robot OR Turntable_Bypassed) AND All_Sensors_Off AND Weld_Robots_Clear);
			Valve2FB.In_Auto_SideB_Command:= Unclamp_Step.1;
		ELSE
			Valve2FB.In_Auto_SideA_Command:= FALSE;
			Valve2FB.In_Auto_SideB_Command:= TRUE;
		END_IF

	(*Valve 3, Model 524 ONLY*)
	(*Slide #4, 11*)
		Valve3FB
			(
			Enable_Motion:= Enable_Motion,
			Enable_Latch:= TRUE,					(*Enabling Runs Valve as detent type (maintained solenoids*)
			Enable_SideA_PreCharge:= FALSE,		(*Enabling Turns Side A PreCharge Active, reset when Side B is energized in Auto*)
			Enable_SideB_PreCharge:= FALSE,		(*Enabling Turns Side B PreCharge Active, reset when Side A is energized in Auto*)
			PreCharge_Time:= T#0.10S,
			Enable_Auto_Commands:= In_Auto,
			Enable_Manual_Commands:= In_Manual AND (All_Robots_Clear OR TurntableB_At_Robot),  (*TLK ADDED OR*)
			In_Manual_SideA_Command:= Discrete_In.ManReqs.4,
			In_Manual_SideB_Command:= (Discrete_In.ManReqs.5 OR Discrete_In.Go_Home),
			SideA_Indicator:= Slide4ADVD AND Slide11ADVD,
			SideB_Indicator:= (Slide4RETD AND Slide11RETD) OR Manual_Ind_HomePrompt,
			TurnOn_SideA_SOL=> N100.Q.4,
			TurnOn_SideB_SOL=> N100.Q.5,
			TurnOn_SideA_Indicator=> Manual_Indicators1.4,
			TurnOn_SideB_Indicator=> Manual_Indicators1.5
			 );
	IF (Model_ID=2) THEN
			Valve3FB.In_Auto_SideA_Command:= Clamp_Step.3 AND NOT Unclamp_Step.2;
			Valve3FB.In_Auto_SideB_Command:= Unclamp_Step.2
										OR ((TurntableA_At_Robot OR Turntable_Bypassed) AND All_Sensors_Off AND Weld_Robots_Clear);
		ELSE
			Valve3FB.In_Auto_SideA_Command:= FALSE;
			Valve3FB.In_Auto_SideB_Command:= TRUE;
		END_IF

	(*Valve 4, Model 543 ONLY*)
	(*Clamp #8, 19*)
		Valve4FB
			(
			Enable_Motion:= Enable_Motion,
			Enable_Latch:= TRUE,					(*Enabling Runs Valve as detent type (maintained solenoids*)
			Enable_SideA_PreCharge:= FALSE,		(*Enabling Turns Side A PreCharge Active, reset when Side B is energized in Auto*)
			Enable_SideB_PreCharge:= FALSE,		(*Enabling Turns Side B PreCharge Active, reset when Side A is energized in Auto*)
			PreCharge_Time:= T#0.10S,
			Enable_Auto_Commands:= In_Auto,
			Enable_Manual_Commands:= In_Manual AND (All_Robots_Clear OR TurntableB_At_Robot),  (*TLK ADDED OR*)
			In_Manual_SideA_Command:= Discrete_In.ManReqs.6,
			In_Manual_SideB_Command:= (Discrete_In.ManReqs.7 OR Discrete_In.Go_Home),
			SideA_Indicator:= Clamp8ADVD AND Clamp19ADVD,
			SideB_Indicator:= (Clamp8RETD AND Clamp19RETD) OR Manual_Ind_HomePrompt,
			TurnOn_SideA_SOL=> N100.Q.6,
			TurnOn_SideB_SOL=> N100.Q.7,
			TurnOn_SideA_Indicator=> Manual_Indicators1.6,
			TurnOn_SideB_Indicator=> Manual_Indicators1.7
			 );
	IF (Model_ID=3) THEN
			Valve4FB.In_Auto_SideA_Command:= Clamp_Step.1 AND NOT Unclamp_Step.0;
			Valve4FB.In_Auto_SideB_Command:= Unclamp_Step.0
										OR ((TurntableA_At_Robot OR Turntable_Bypassed) AND All_Sensors_Off AND Weld_Robots_Clear);
		ELSE
			Valve4FB.In_Auto_SideA_Command:= FALSE;
			Valve4FB.In_Auto_SideB_Command:= TRUE;
		END_IF

	(*Valve 5, Model 543 ONLY*)
	(*Pin #6, 14*)
		Valve5FB
			(
			Enable_Motion:= Enable_Motion,
			Enable_Latch:= TRUE,					(*Enabling Runs Valve as detent type (maintained solenoids*)
			Enable_SideA_PreCharge:= FALSE,		(*Enabling Turns Side A PreCharge Active, reset when Side B is energized in Auto*)
			Enable_SideB_PreCharge:= FALSE,		(*Enabling Turns Side B PreCharge Active, reset when Side A is energized in Auto*)
			PreCharge_Time:= T#0.10S,
			Enable_Auto_Commands:= In_Auto,
			Enable_Manual_Commands:= In_Manual AND (All_Robots_Clear OR TurntableB_At_Robot),  (*TLK ADDED OR*)
			In_Manual_SideA_Command:= (Discrete_In.ManReqs.8 OR (Discrete_In.Go_Home AND (Model_ID = 3))),
			In_Manual_SideB_Command:= (Discrete_In.ManReqs.9 OR (Discrete_In.Go_Home AND (Model_ID <> 3))),
			SideA_Indicator:=  Pin6ADVD AND Pin14ADVD,
			SideB_Indicator:= (Pin6RETD AND Pin14RETD) OR Manual_Ind_HomePrompt,
			TurnOn_SideA_SOL=> N100.Q.8,
			TurnOn_SideB_SOL=> N100.Q.9,
			TurnOn_SideA_Indicator=> Manual_Indicators1.8,
			TurnOn_SideB_Indicator=> Manual_Indicators1.9
			 );
	IF (Model_ID=3) THEN		 
			Valve5FB.In_Auto_SideA_Command:= Clamp_Step.0 AND NOT Unclamp_Step.1
										OR ((TurntableA_At_Robot OR Turntable_Bypassed) AND All_Sensors_Off AND Weld_Robots_Clear);
			Valve5FB.In_Auto_SideB_Command:= Unclamp_Step.1;
		ELSE
			Valve5FB.In_Auto_SideA_Command:= FALSE;
			Valve5FB.In_Auto_SideB_Command:= TRUE;
		END_IF

	(*Valve 6, Model 543 ONLY*)
	(*Swing #1, 3*)
		Valve6FB
			(
			Enable_Motion:= Enable_Motion,
			Enable_Latch:= TRUE,					(*Enabling Runs Valve as detent type (maintained solenoids*)
			Enable_SideA_PreCharge:= FALSE,		(*Enabling Turns Side A PreCharge Active, reset when Side B is energized in Auto*)
			Enable_SideB_PreCharge:= FALSE,		(*Enabling Turns Side B PreCharge Active, reset when Side A is energized in Auto*)
			PreCharge_Time:= T#0.10S,
			Enable_Auto_Commands:= In_Auto,
			Enable_Manual_Commands:= In_Manual AND (All_Robots_Clear OR TurntableB_At_Robot),  (*TLK ADDED OR*)
			In_Manual_SideA_Command:= Discrete_In.ManReqs.10,
			In_Manual_SideB_Command:= (Discrete_In.ManReqs.11 OR Discrete_In.Go_Home),
			SideA_Indicator:= Swing1ADVD AND Swing3ADVD,
			SideB_Indicator:= (Swing1RETD AND Swing3RETD) OR Manual_Ind_HomePrompt,
			TurnOn_SideA_SOL=> N100.Q.10,
			TurnOn_SideB_SOL=> N100.Q.11,
			TurnOn_SideA_Indicator=> Manual_Indicators1.10,
			TurnOn_SideB_Indicator=> Manual_Indicators1.11
			 );
	IF (Model_ID=3) THEN
			Valve6FB.In_Auto_SideA_Command:= Clamp_Step.3 AND NOT Unclamp_Step.2;
			Valve6FB.In_Auto_SideB_Command:= Unclamp_Step.2
										OR ((TurntableA_At_Robot OR Turntable_Bypassed) AND All_Sensors_Off AND Weld_Robots_Clear);
		ELSE
			Valve6FB.In_Auto_SideA_Command:= FALSE;
			Valve6FB.In_Auto_SideB_Command:= TRUE;
		END_IF

	(*Valve 7, Common*)
	(*Clamp #3, 18 - Manual Clamps*)
		Valve7FB
			(
			Enable_Motion:= Enable_Motion,
			Enable_Latch:= (TurnTable_WorkingOK OR TurnTableA_At_Robot),					(*Enabling Runs Valve as detent type (maintained solenoids*)
			Enable_SideA_PreCharge:= FALSE,		(*Enabling Turns Side A PreCharge Active, reset when Side B is energized in Auto*)
			Enable_SideB_PreCharge:= FALSE,		(*Enabling Turns Side B PreCharge Active, reset when Side A is energized in Auto*)
			PreCharge_Time:= T#0.10S,
			Enable_Auto_Commands:= In_Auto,
			Enable_Manual_Commands:= In_Manual AND (All_Robots_Clear OR TurntableB_At_Robot),  (*TLK ADDED OR*)
			In_Manual_SideA_Command:= Discrete_In.ManReqs.12,
			In_Manual_SideB_Command:= (Discrete_In.ManReqs.13 OR Discrete_In.Go_Home),
			SideA_Indicator:= Clamp3ADVD AND Clamp18ADVD,
			SideB_Indicator:= (Clamp3RETD AND Clamp18RETD) OR Manual_Ind_HomePrompt,
			TurnOn_SideA_SOL=> N100.Q.12,
			TurnOn_SideB_SOL=> N100.Q.13,
			TurnOn_SideA_Indicator=> Manual_Indicators1.12,
			TurnOn_SideB_Indicator=> Manual_Indicators1.13
			 );
		Valve7FB.In_Auto_SideA_Command:= Clamp_Step.1 AND NOT Unclamp_Step.0;
		Valve7FB.In_Auto_SideB_Command:= Unclamp_Step.0
										OR ((TurntableB_At_Robot OR Turntable_Bypassed) AND All_Sensors_Off AND Weld_Robots_Clear);


	(*Valve 8, Common*)
	(*Pin #1-4, 7, 9, 16-18, Slide #10*)
		Valve8FB
			(
			Enable_Motion:= Enable_Motion,
			Enable_Latch:= TRUE,					(*Enabling Runs Valve as detent type (maintained solenoids*)
			Enable_SideA_PreCharge:= FALSE,		(*Enabling Turns Side A PreCharge Active, reset when Side B is energized in Auto*)
			Enable_SideB_PreCharge:= FALSE,		(*Enabling Turns Side B PreCharge Active, reset when Side A is energized in Auto*)
			PreCharge_Time:= T#0.10S,
			Enable_Auto_Commands:= In_Auto,
			Enable_Manual_Commands:= In_Manual AND (All_Robots_Clear OR TurntableB_At_Robot),  (*TLK ADDED OR*)
			In_Manual_SideA_Command:= (Discrete_In.ManReqs.14 OR Discrete_In.Go_Home),
			In_Manual_SideB_Command:= Discrete_In.ManReqs.15,
			SideA_Indicator:= (Pin1ADVD AND Pin2ADVD AND Pin3ADVD AND Pin4ADVD AND Pin7ADVD AND Pin9ADVD AND Pin16ADVD AND Pin17ADVD AND Pin18ADVD AND Slide10ADVD) OR Manual_Ind_HomePrompt,
			SideB_Indicator:= Pin1RETD AND Pin2RETD AND Pin3RETD AND Pin4RETD AND Pin7RETD AND Pin9RETD AND Pin16RETD AND Pin17RETD AND Pin18RETD AND Slide10RETD,
			TurnOn_SideA_SOL=> N100.Q.14,
			TurnOn_SideB_SOL=> N100.Q.15,
			TurnOn_SideA_Indicator=> Manual_Indicators1.14,
			TurnOn_SideB_Indicator=> Manual_Indicators1.15
			 );
		Valve8FB.In_Auto_SideA_Command:= Clamp_Step.0 AND NOT Unclamp_Step.1
										OR ((TurntableA_At_Robot OR Turntable_Bypassed) AND All_Sensors_Off AND Weld_Robots_Clear);
		Valve8FB.In_Auto_SideB_Command:= Unclamp_Step.1;


	(*Valve 9, Common*)
	(*Clamp #1, 2, 4, 5, 10, 14, 21, 22*)
		Valve9FB
			(
			Enable_Motion:= Enable_Motion,
			Enable_Latch:= TRUE,					(*Enabling Runs Valve as detent type (maintained solenoids*)
			Enable_SideA_PreCharge:= FALSE,		(*Enabling Turns Side A PreCharge Active, reset when Side B is energized in Auto*)
			Enable_SideB_PreCharge:= FALSE,		(*Enabling Turns Side B PreCharge Active, reset when Side A is energized in Auto*)
			PreCharge_Time:= T#0.10S,
			Enable_Auto_Commands:= In_Auto,
			Enable_Manual_Commands:= In_Manual AND (All_Robots_Clear OR TurntableB_At_Robot),  (*TLK ADDED OR*)
			In_Manual_SideA_Command:= Discrete_In.ManReqs.16,
			In_Manual_SideB_Command:= (Discrete_In.ManReqs.17 OR Discrete_In.Go_Home),
			SideA_Indicator:= Clamp1ADVD AND Clamp2ADVD AND Clamp4ADVD AND Clamp5ADVD AND Clamp10ADVD AND Clamp14ADVD AND Clamp21ADVD AND Clamp22ADVD,
			SideB_Indicator:= (Clamp1RETD AND Clamp2RETD AND Clamp4RETD AND Clamp5RETD AND Clamp10RETD AND Clamp14RETD AND Clamp21RETD AND Clamp22RETD) OR Manual_Ind_HomePrompt,
			TurnOn_SideA_SOL=> N100.Q.16,
			TurnOn_SideB_SOL=> N100.Q.17,
			TurnOn_SideA_Indicator=> Manual_Indicators1.16,
			TurnOn_SideB_Indicator=> Manual_Indicators1.17
			 );
		Valve9FB.In_Auto_SideA_Command:= Clamp_Step.1 AND NOT Unclamp_Step.0;
		Valve9FB.In_Auto_SideB_Command:= Unclamp_Step.0
										OR ((TurntableA_At_Robot OR Turntable_Bypassed) AND All_Sensors_Off AND Weld_Robots_Clear);


	(*Valve 10, Common*)
	(*Pin #8, 10-13, Slide #1, 2, 13, 14*)
		Valve10FB
			(
			Enable_Motion:= Enable_Motion,
			Enable_Latch:= TRUE,					(*Enabling Runs Valve as detent type (maintained solenoids*)
			Enable_SideA_PreCharge:= FALSE,		(*Enabling Turns Side A PreCharge Active, reset when Side B is energized in Auto*)
			Enable_SideB_PreCharge:= FALSE,		(*Enabling Turns Side B PreCharge Active, reset when Side A is energized in Auto*)
			PreCharge_Time:= T#0.10S,
			Enable_Auto_Commands:= In_Auto,
			Enable_Manual_Commands:= In_Manual AND (All_Robots_Clear OR TurntableB_At_Robot),  (*TLK ADDED OR*)
			In_Manual_SideA_Command:= (Discrete_In.ManReqs.18 OR Discrete_In.Go_Home),
			In_Manual_SideB_Command:= Discrete_In.ManReqs.19,
			SideA_Indicator:= (Pin8ADVD AND Pin10ADVD AND Pin11ADVD AND Pin12ADVD AND Pin13ADVD AND Slide1ADVD AND Slide2ADVD AND Slide13ADVD AND Slide14ADVD) OR Manual_Ind_HomePrompt,
			SideB_Indicator:= Pin8RETD AND Pin10RETD AND Pin11RETD AND Pin12RETD AND Pin13RETD AND Slide1RETD AND Slide2RETD AND Slide13RETD AND Slide14RETD,
			TurnOn_SideA_SOL=> N100.Q.18,
			TurnOn_SideB_SOL=> N100.Q.19,
			TurnOn_SideA_Indicator=> Manual_Indicators1.18,
			TurnOn_SideB_Indicator=> Manual_Indicators1.19
			 );
		Valve10FB.In_Auto_SideA_Command:= Clamp_Step.0 AND NOT Unclamp_Step.1
										OR ((TurntableA_At_Robot OR Turntable_Bypassed) AND All_Sensors_Off AND Weld_Robots_Clear);
		Valve10FB.In_Auto_SideB_Command:= Unclamp_Step.1;


	(*Valve 11, Common*)
	(*Clamp #9, 12, 13, 16*)
		Valve11FB
			(
			Enable_Motion:= Enable_Motion,
			Enable_Latch:= TRUE,					(*Enabling Runs Valve as detent type (maintained solenoids*)
			Enable_SideA_PreCharge:= FALSE,		(*Enabling Turns Side A PreCharge Active, reset when Side B is energized in Auto*)
			Enable_SideB_PreCharge:= FALSE,		(*Enabling Turns Side B PreCharge Active, reset when Side A is energized in Auto*)
			PreCharge_Time:= T#0.10S,
			Enable_Auto_Commands:= In_Auto,
			Enable_Manual_Commands:= In_Manual AND (All_Robots_Clear OR TurntableB_At_Robot),  (*TLK ADDED OR*)
			In_Manual_SideA_Command:= Discrete_In.ManReqs.20,
			In_Manual_SideB_Command:= (Discrete_In.ManReqs.21 OR Discrete_In.Go_Home),
			SideA_Indicator:= Clamp9ADVD AND Clamp12ADVD AND Clamp13ADVD AND Clamp16ADVD,
			SideB_Indicator:= (Clamp9RETD AND Clamp12RETD AND Clamp13RETD AND Clamp16RETD) OR Manual_Ind_HomePrompt,
			TurnOn_SideA_SOL=> N100.Q.20,
			TurnOn_SideB_SOL=> N100.Q.21,
			TurnOn_SideA_Indicator=> Manual_Indicators1.20,
			TurnOn_SideB_Indicator=> Manual_Indicators1.21
			 );
		Valve11FB.In_Auto_SideA_Command:= Clamp_Step.1 AND NOT Unclamp_Step.0;
		Valve11FB.In_Auto_SideB_Command:= Unclamp_Step.0
										OR ((TurntableA_At_Robot OR Turntable_Bypassed) AND All_Sensors_Off AND Weld_Robots_Clear);


	(*Valve 12, Common*)
	(*Slide #3, 5, 7-9, 12, Swing #2*)
		Valve12FB
			(
			Enable_Motion:= Enable_Motion,
			Enable_Latch:= TRUE,					(*Enabling Runs Valve as detent type (maintained solenoids*)
			Enable_SideA_PreCharge:= FALSE,		(*Enabling Turns Side A PreCharge Active, reset when Side B is energized in Auto*)
			Enable_SideB_PreCharge:= FALSE,		(*Enabling Turns Side B PreCharge Active, reset when Side A is energized in Auto*)
			PreCharge_Time:= T#0.10S,
			Enable_Auto_Commands:= In_Auto,
			Enable_Manual_Commands:= In_Manual AND (All_Robots_Clear OR TurntableB_At_Robot),  (*TLK ADDED OR*)
			In_Manual_SideA_Command:= Discrete_In.ManReqs.22,
			In_Manual_SideB_Command:= (Discrete_In.ManReqs.23 OR Discrete_In.Go_Home),
			SideA_Indicator:= Slide3ADVD AND Slide5ADVD AND Slide7ADVD AND Slide8ADVD AND Slide9ADVD AND Slide12ADVD AND Swing2ADVD,
			SideB_Indicator:= (Slide3RETD AND Slide5RETD AND Slide7RETD AND Slide8RETD AND Slide9RETD AND Slide12RETD AND Swing2RETD) OR Manual_Ind_HomePrompt,
			TurnOn_SideA_SOL=> N100.Q.22,
			TurnOn_SideB_SOL=> N100.Q.23,
			TurnOn_SideA_Indicator=> Manual_Indicators1.22,
			TurnOn_SideB_Indicator=> Manual_Indicators1.23
			 );
		Valve12FB.In_Auto_SideA_Command:= Clamp_Step.3 AND NOT Unclamp_Step.2;
		Valve12FB.In_Auto_SideB_Command:= Unclamp_Step.2
										OR ((TurntableA_At_Robot OR Turntable_Bypassed) AND All_Sensors_Off AND Weld_Robots_Clear);


	(*Valve 13, Common*)
	(*Clamp #7, 11, 15, 17*)
		Valve13FB
			(
			Enable_Motion:= Enable_Motion,
			Enable_Latch:= TRUE,					(*Enabling Runs Valve as detent type (maintained solenoids*)
			Enable_SideA_PreCharge:= FALSE,		(*Enabling Turns Side A PreCharge Active, reset when Side B is energized in Auto*)
			Enable_SideB_PreCharge:= FALSE,		(*Enabling Turns Side B PreCharge Active, reset when Side A is energized in Auto*)
			PreCharge_Time:= T#0.10S,
			Enable_Auto_Commands:= In_Auto,
			Enable_Manual_Commands:= In_Manual AND (All_Robots_Clear OR TurntableB_At_Robot),  (*TLK ADDED OR*)
			In_Manual_SideA_Command:= Discrete_In.ManReqs.24,
			In_Manual_SideB_Command:= (Discrete_In.ManReqs.25 OR Discrete_In.Go_Home),
			SideA_Indicator:= Clamp7ADVD AND Clamp11ADVD AND Clamp15ADVD AND Clamp17ADVD,
			SideB_Indicator:= (Clamp7RETD AND Clamp11RETD AND Clamp15RETD AND Clamp17RETD) OR Manual_Ind_HomePrompt,
			TurnOn_SideA_SOL=> N100.Q.24,
			TurnOn_SideB_SOL=> N100.Q.25,
			TurnOn_SideA_Indicator=> Manual_Indicators1.24,
			TurnOn_SideB_Indicator=> Manual_Indicators1.25
			 );
		Valve13FB.In_Auto_SideA_Command:= Clamp_Step.2 AND NOT Unclamp_Step.3;
		Valve13FB.In_Auto_SideB_Command:= Unclamp_Step.3
										OR ((TurntableA_At_Robot OR Turntable_Bypassed) AND All_Sensors_Off AND Weld_Robots_Clear);	
		
		
	(*Valve 14, A+B*)
	(*Locks*)
		Valve14FB
			(
			Enable_Motion:= Enable_Motion ,
			Enable_Latch:= FALSE,					(*Enabling Runs Valve as detent type (maintained solenoids*)
			Enable_SideA_PreCharge:= FALSE,		(*Enabling Turns Side A PreCharge Active, reset when Side B is energized in Auto*)
			Enable_SideB_PreCharge:= FALSE,		(*Enabling Turns Side B PreCharge Active, reset when Side A is energized in Auto*)
			PreCharge_Time:= T#0.10S,
			Enable_Auto_Commands:= In_Auto,
			Enable_Manual_Commands:= In_Manual AND (All_Robots_Clear OR TurntableB_At_Robot),
			In_Manual_SideA_Command:= Discrete_In.ManReqs.26,
			In_Manual_SideB_Command:= Discrete_In.ManReqs.27 
										OR (N100.Q.5 AND NOT (Slide4RETD AND Slide11RETD)) 
										OR (N100.Q.15 AND NOT Slide10RETD) 
										OR (N100.Q.19 AND NOT (Slide1RETD AND Slide2RETD AND Slide13RETD AND Slide14RETD))
										OR (N100.Q.23 AND NOT (Slide3RETD AND Slide5RETD AND Slide7RETD AND Slide8RETD AND Slide9RETD AND Slide12RETD))
										OR (N100.Q.28 AND NOT Slide6RETD)
										OR (N100.Q.4 AND NOT (Slide4ADVD AND Slide11ADVD)) 
										OR (N100.Q.14 AND NOT Slide10ADVD) 
										OR (N100.Q.18 AND NOT (Slide1ADVD AND Slide2ADVD AND Slide13ADVD AND Slide14ADVD))
										OR (N100.Q.22 AND NOT (Slide3ADVD AND Slide5ADVD AND Slide7ADVD AND Slide8ADVD AND Slide9ADVD AND Slide12ADVD))
										OR (N100.Q.28 AND NOT Slide6ADVD),
			SideA_Indicator:= FALSE,
			SideB_Indicator:= FALSE,
			TurnOn_SideA_SOL=> N100.Q.26,
			TurnOn_SideB_SOL=> N100.Q.27,
			TurnOn_SideA_Indicator=> Manual_Indicators1.26,
			TurnOn_SideB_Indicator=> Manual_Indicators1.27
			 );
		Valve14FB.In_Auto_SideA_Command:= NOT Valve14FB.In_Auto_SideB_Command;
		Valve14FB.In_Auto_SideB_Command:= (N100.Q.5 AND NOT (Slide4RETD AND Slide11RETD)) 
										OR (N100.Q.15 AND NOT Slide10RETD) 
										OR (N100.Q.19 AND NOT (Slide1RETD AND Slide2RETD AND Slide13RETD AND Slide14RETD))
										OR (N100.Q.23 AND NOT (Slide3RETD AND Slide5RETD AND Slide7RETD AND Slide8RETD AND Slide9RETD AND Slide12RETD))
										OR (N100.Q.29 AND NOT Slide6RETD)
										OR (N100.Q.4 AND NOT (Slide4ADVD AND Slide11ADVD)) 
										OR (N100.Q.14 AND NOT Slide10ADVD) 
										OR (N100.Q.18 AND NOT (Slide1ADVD AND Slide2ADVD AND Slide13ADVD AND Slide14ADVD))
										OR (N100.Q.22 AND NOT (Slide3ADVD AND Slide5ADVD AND Slide7ADVD AND Slide8ADVD AND Slide9ADVD AND Slide12ADVD))
										OR (N100.Q.28 AND NOT Slide6ADVD);



	(*Valve 15, A+B*)
	(*Slide #6*)
		Valve15FB
			(
			Enable_Motion:= Enable_Motion ,
			Enable_Latch:= TRUE,					(*Enabling Runs Valve as detent type (maintained solenoids*)
			Enable_SideA_PreCharge:= FALSE,		(*Enabling Turns Side A PreCharge Active, reset when Side B is energized in Auto*)
			Enable_SideB_PreCharge:= FALSE,		(*Enabling Turns Side B PreCharge Active, reset when Side A is energized in Auto*)
			PreCharge_Time:= T#0.10S,
			Enable_Auto_Commands:= In_Auto,
			Enable_Manual_Commands:= In_Manual AND (All_Robots_Clear OR TurntableB_At_Robot),  (*TLK ADDED OR*)
			In_Manual_SideA_Command:= Discrete_In.ManReqs.28,
			In_Manual_SideB_Command:= Discrete_In.ManReqs.29,
			SideA_Indicator:= Slide6ADVD,
			SideB_Indicator:= Slide6RETD,
			TurnOn_SideA_SOL=> N100.Q.28,
			TurnOn_SideB_SOL=> N100.Q.29,
			TurnOn_SideA_Indicator=> Manual_Indicators1.28,
			TurnOn_SideB_Indicator=> Manual_Indicators1.29
			 );
		Valve15FB.In_Auto_SideA_Command:= Clamp_Step.3 AND NOT Unclamp_Step.2;
		Valve15FB.In_Auto_SideB_Command:= ((TurntableA_At_Robot OR Turntable_Bypassed) AND All_Sensors_Off AND Weld_Robots_Clear);
		
		
(*--------------------------------------------------------------------------------------------------------------------------------------------*)		
(*                                                           Spare Valves                                                                     *)
(*--------------------------------------------------------------------------------------------------------------------------------------------*)


	(*Valve 16, A+B*)
	(*spare*)
		Valve16FB
			(
			Enable_Motion:= Enable_Motion ,
			Enable_Latch:= TRUE,					(*Enabling Runs Valve as detent type (maintained solenoids*)
			Enable_SideA_PreCharge:= FALSE,		(*Enabling Turns Side A PreCharge Active, reset when Side B is energized in Auto*)
			Enable_SideB_PreCharge:= FALSE,		(*Enabling Turns Side B PreCharge Active, reset when Side A is energized in Auto*)
			PreCharge_Time:= T#0.10S,
			Enable_Auto_Commands:= In_Auto,
			Enable_Manual_Commands:= In_Manual AND (All_Robots_Clear OR TurntableB_At_Robot),  (*TLK ADDED OR*)
			In_Manual_SideA_Command:= Discrete_In.ManReqs.30,
			In_Manual_SideB_Command:= Discrete_In.ManReqs.31,
			SideA_Indicator:= FALSE,
			SideB_Indicator:= FALSE,
			TurnOn_SideA_SOL=> N100.Q.30,
			TurnOn_SideB_SOL=> N100.Q.31,
			TurnOn_SideA_Indicator=> Manual_Indicators1.30,
			TurnOn_SideB_Indicator=> Manual_Indicators1.31
			 );
		Valve16FB.In_Auto_SideA_Command:= FALSE;
		Valve16FB.In_Auto_SideB_Command:= FALSE;


























(*end*)
END_ACTION

ACTION ValveBank2:


(*+++++++++++THIS AREA IS CUSTOM PER INSTALLATION AND WILL HAVE TO BE MODIFIED PER +++++++++++++*)
(*+++++++++++THIS AREA IS CUSTOM PER INSTALLATION AND WILL HAVE TO BE MODIFIED PER +++++++++++++*)
(*+++++++++++THIS AREA IS CUSTOM PER INSTALLATION AND WILL HAVE TO BE MODIFIED PER +++++++++++++*)

(*+++++++++++VALVE BANK 2 +++++++++++++*)
(*+++++++++++VALVE BANK 2 +++++++++++++*)
(*+++++++++++VALVE BANK 2 +++++++++++++*)


	(*Valve 17, A+B*)
	(*spare*)
		Valve17FB
			(
			Enable_Motion:= Enable_Motion ,
			Enable_Latch:= TRUE,					(*Enabling Runs Valve as detent type (maintained solenoids*)
			Enable_SideA_PreCharge:= FALSE,		(*Enabling Turns Side A PreCharge Active, reset when Side B is energized in Auto*)
			Enable_SideB_PreCharge:= FALSE,		(*Enabling Turns Side B PreCharge Active, reset when Side A is energized in Auto*)
			PreCharge_Time:= T#0.1S,
			Enable_Auto_Commands:= In_Auto,
			Enable_Manual_Commands:= In_Manual AND All_Robots_Clear,
			In_Manual_SideA_Command:= Discrete_In.ManReqs2.0,
			In_Manual_SideB_Command:= (Discrete_In.ManReqs2.1 OR Discrete_In.Go_Home),
			SideA_Indicator:= FALSE,
			SideB_Indicator:= FALSE,
			TurnOn_SideA_SOL=> N101.Q.0,
			TurnOn_SideB_SOL=> N101.Q.1,
			TurnOn_SideA_Indicator=> Manual_Indicators2.0,
			TurnOn_SideB_Indicator=> Manual_Indicators2.1
			 );
		Valve17FB.In_Auto_SideA_Command:= FALSE;
		Valve17FB.In_Auto_SideB_Command:= FALSE;


	(*Valve 18, A+B*)
	(*spare*)
		Valve18FB
			(
			Enable_Motion:= Enable_Motion ,
			Enable_Latch:= TRUE,					(*Enabling Runs Valve as detent type (maintained solenoids*)
			Enable_SideA_PreCharge:= FALSE,		(*Enabling Turns Side A PreCharge Active, reset when Side B is energized in Auto*)
			Enable_SideB_PreCharge:= FALSE,		(*Enabling Turns Side B PreCharge Active, reset when Side A is energized in Auto*)
			PreCharge_Time:= T#0.10S,
			Enable_Auto_Commands:= In_Auto,
			Enable_Manual_Commands:= In_Manual AND All_Robots_Clear,
			In_Manual_SideA_Command:= Discrete_In.ManReqs2.2,
			In_Manual_SideB_Command:= Discrete_In.ManReqs2.3,
			SideA_Indicator:= FALSE,
			SideB_Indicator:= FALSE,
			TurnOn_SideA_SOL=> N101.Q.2,
			TurnOn_SideB_SOL=> N101.Q.3,
			TurnOn_SideA_Indicator=> Manual_Indicators2.2,
			TurnOn_SideB_Indicator=> Manual_Indicators2.3
			 );
		Valve18FB.In_Auto_SideA_Command:= FALSE;
		Valve18FB.In_Auto_SideB_Command:= FALSE;

	(*Valve 19, A+B*)
	(*spare*)
		Valve19FB
			(
			Enable_Motion:= Enable_Motion ,
			Enable_Latch:= TRUE,					(*Enabling Runs Valve as detent type (maintained solenoids*)
			Enable_SideA_PreCharge:= FALSE,		(*Enabling Turns Side A PreCharge Active, reset when Side B is energized in Auto*)
			Enable_SideB_PreCharge:= FALSE,		(*Enabling Turns Side B PreCharge Active, reset when Side A is energized in Auto*)
			PreCharge_Time:= T#0.10S,
			Enable_Auto_Commands:= In_Auto,
			Enable_Manual_Commands:= In_Manual AND All_Robots_Clear,
			In_Manual_SideA_Command:= Discrete_In.ManReqs2.4,
			In_Manual_SideB_Command:= Discrete_In.ManReqs2.5,
			SideA_Indicator:= FALSE,
			SideB_Indicator:= FALSE,
			TurnOn_SideA_SOL=> N101.Q.4,
			TurnOn_SideB_SOL=> N101.Q.5,
			TurnOn_SideA_Indicator=> Manual_Indicators2.4,
			TurnOn_SideB_Indicator=> Manual_Indicators2.5
			 );
		Valve19FB.In_Auto_SideA_Command:= FALSE;
		Valve19FB.In_Auto_SideB_Command:= FALSE;


	(*Valve 20, A+B*)
	(*spare*)
		Valve20FB
			(
			Enable_Motion:= Enable_Motion ,
			Enable_Latch:= TRUE,					(*Enabling Runs Valve as detent type (maintained solenoids*)
			Enable_SideA_PreCharge:= FALSE,		(*Enabling Turns Side A PreCharge Active, reset when Side B is energized in Auto*)
			Enable_SideB_PreCharge:= FALSE,		(*Enabling Turns Side B PreCharge Active, reset when Side A is energized in Auto*)
			PreCharge_Time:= T#0.10S,
			Enable_Auto_Commands:= In_Auto,
			Enable_Manual_Commands:= In_Manual AND All_Robots_Clear,
			In_Manual_SideA_Command:= Discrete_In.ManReqs2.6,
			In_Manual_SideB_Command:= Discrete_In.ManReqs2.7,
			SideA_Indicator:= FALSE,
			SideB_Indicator:= FALSE,
			TurnOn_SideA_SOL=> N101.Q.6,
			TurnOn_SideB_SOL=> N101.Q.7,
			TurnOn_SideA_Indicator=> Manual_Indicators2.6,
			TurnOn_SideB_Indicator=> Manual_Indicators2.7
			 );
		Valve20FB.In_Auto_SideA_Command:= FALSE;
		Valve20FB.In_Auto_SideB_Command:= FALSE;


	(*Valve 21, A+B*)
	(*spare*)
		Valve21FB
			(
			Enable_Motion:= Enable_Motion ,
			Enable_Latch:= TRUE,					(*Enabling Runs Valve as detent type (maintained solenoids*)
			Enable_SideA_PreCharge:= FALSE,		(*Enabling Turns Side A PreCharge Active, reset when Side B is energized in Auto*)
			Enable_SideB_PreCharge:= FALSE,		(*Enabling Turns Side B PreCharge Active, reset when Side A is energized in Auto*)
			PreCharge_Time:= T#0.10S,
			Enable_Auto_Commands:= In_Auto,
			Enable_Manual_Commands:= In_Manual AND All_Robots_Clear,
			In_Manual_SideA_Command:= Discrete_In.ManReqs2.8,
			In_Manual_SideB_Command:= Discrete_In.ManReqs2.9,
			SideA_Indicator:= FALSE,
			SideB_Indicator:= FALSE,
			TurnOn_SideA_SOL=> N101.Q.8,
			TurnOn_SideB_SOL=> N101.Q.9,
			TurnOn_SideA_Indicator=> Manual_Indicators2.8,
			TurnOn_SideB_Indicator=> Manual_Indicators2.9
			 );
		Valve21FB.In_Auto_SideA_Command:= FALSE;
		Valve21FB.In_Auto_SideB_Command:= FALSE;


	(*Valve 22, A+B*)
	(*spare*)
		Valve22FB
			(
			Enable_Motion:= Enable_Motion ,
			Enable_Latch:= TRUE,					(*Enabling Runs Valve as detent type (maintained solenoids*)
			Enable_SideA_PreCharge:= FALSE,		(*Enabling Turns Side A PreCharge Active, reset when Side B is energized in Auto*)
			Enable_SideB_PreCharge:= FALSE,		(*Enabling Turns Side B PreCharge Active, reset when Side A is energized in Auto*)
			PreCharge_Time:= T#0.10S,
			Enable_Auto_Commands:= In_Auto,
			Enable_Manual_Commands:= In_Manual AND All_Robots_Clear,
			In_Manual_SideA_Command:= Discrete_In.ManReqs2.10,
			In_Manual_SideB_Command:= Discrete_In.ManReqs2.11,
			SideA_Indicator:= FALSE,
			SideB_Indicator:= FALSE,
			TurnOn_SideA_SOL=> N101.Q.10,
			TurnOn_SideB_SOL=> N101.Q.11,
			TurnOn_SideA_Indicator=> Manual_Indicators2.10,
			TurnOn_SideB_Indicator=> Manual_Indicators2.11
			 );
		Valve22FB.In_Auto_SideA_Command:= FALSE;
		Valve22FB.In_Auto_SideB_Command:= FALSE;


	(*Valve 23, A+B*)
	(*spare*)
		Valve23FB
			(
			Enable_Motion:= Enable_Motion ,
			Enable_Latch:= TRUE,					(*Enabling Runs Valve as detent type (maintained solenoids*)
			Enable_SideA_PreCharge:= FALSE,		(*Enabling Turns Side A PreCharge Active, reset when Side B is energized in Auto*)
			Enable_SideB_PreCharge:= FALSE,		(*Enabling Turns Side B PreCharge Active, reset when Side A is energized in Auto*)
			PreCharge_Time:= T#0.10S,
			Enable_Auto_Commands:= In_Auto,
			Enable_Manual_Commands:= In_Manual AND All_Robots_Clear,
			In_Manual_SideA_Command:= Discrete_In.ManReqs2.12,
			In_Manual_SideB_Command:= Discrete_In.ManReqs2.13,
			SideA_Indicator:= FALSE,
			SideB_Indicator:= FALSE,
			TurnOn_SideA_SOL=> N101.Q.12,
			TurnOn_SideB_SOL=> N101.Q.13,
			TurnOn_SideA_Indicator=> Manual_Indicators2.12,
			TurnOn_SideB_Indicator=> Manual_Indicators2.13
			 );
		Valve23FB.In_Auto_SideA_Command:= FALSE;
		Valve23FB.In_Auto_SideB_Command:= FALSE;


	(*Valve 24, A+B*)
	(*spare*)
		Valve24FB
			(
			Enable_Motion:= Enable_Motion ,
			Enable_Latch:= TRUE,					(*Enabling Runs Valve as detent type (maintained solenoids*)
			Enable_SideA_PreCharge:= FALSE,		(*Enabling Turns Side A PreCharge Active, reset when Side B is energized in Auto*)
			Enable_SideB_PreCharge:= FALSE,		(*Enabling Turns Side B PreCharge Active, reset when Side A is energized in Auto*)
			PreCharge_Time:= T#0.10S,
			Enable_Auto_Commands:= In_Auto,
			Enable_Manual_Commands:= In_Manual AND All_Robots_Clear,
			In_Manual_SideA_Command:= Discrete_In.ManReqs2.14,
			In_Manual_SideB_Command:= Discrete_In.ManReqs2.15,
			SideA_Indicator:= FALSE,
			SideB_Indicator:= FALSE,
			TurnOn_SideA_SOL=> N101.Q.14,
			TurnOn_SideB_SOL=> N101.Q.15,
			TurnOn_SideA_Indicator=> Manual_Indicators2.14,
			TurnOn_SideB_Indicator=> Manual_Indicators2.15
			 );
		Valve24FB.In_Auto_SideA_Command:= FALSE;
		Valve24FB.In_Auto_SideB_Command:= FALSE;


	(*Valve 25, A+B*)
	(*spare*)
		Valve25FB
			(
			Enable_Motion:= Enable_Motion ,
			Enable_Latch:= TRUE,					(*Enabling Runs Valve as detent type (maintained solenoids*)
			Enable_SideA_PreCharge:= FALSE,		(*Enabling Turns Side A PreCharge Active, reset when Side B is energized in Auto*)
			Enable_SideB_PreCharge:= FALSE,		(*Enabling Turns Side B PreCharge Active, reset when Side A is energized in Auto*)
			PreCharge_Time:= T#0.10S,
			Enable_Auto_Commands:= In_Auto,
			Enable_Manual_Commands:= In_Manual AND All_Robots_Clear,
			In_Manual_SideA_Command:= Discrete_In.ManReqs2.16,
			In_Manual_SideB_Command:= Discrete_In.ManReqs2.17,
			SideA_Indicator:= FALSE,
			SideB_Indicator:= FALSE,
			TurnOn_SideA_SOL=> N101.Q.16,
			TurnOn_SideB_SOL=> N101.Q.17,
			TurnOn_SideA_Indicator=> Manual_Indicators2.16,
			TurnOn_SideB_Indicator=> Manual_Indicators2.17
			 );
		Valve25FB.In_Auto_SideA_Command:= FALSE;
		Valve25FB.In_Auto_SideB_Command:= FALSE;


	(*Valve 26, A+B*)
	(*spare*)
		Valve26FB
			(
			Enable_Motion:= Enable_Motion ,
			Enable_Latch:= TRUE,					(*Enabling Runs Valve as detent type (maintained solenoids*)
			Enable_SideA_PreCharge:= FALSE,		(*Enabling Turns Side A PreCharge Active, reset when Side B is energized in Auto*)
			Enable_SideB_PreCharge:= FALSE,		(*Enabling Turns Side B PreCharge Active, reset when Side A is energized in Auto*)
			PreCharge_Time:= T#0.10S,
			Enable_Auto_Commands:= In_Auto,
			Enable_Manual_Commands:= In_Manual AND All_Robots_Clear,
			In_Manual_SideA_Command:= Discrete_In.ManReqs2.18,
			In_Manual_SideB_Command:= Discrete_In.ManReqs2.19,
			SideA_Indicator:= FALSE,
			SideB_Indicator:= FALSE,
			TurnOn_SideA_SOL=> N101.Q.18,
			TurnOn_SideB_SOL=> N101.Q.19,
			TurnOn_SideA_Indicator=> Manual_Indicators2.18,
			TurnOn_SideB_Indicator=> Manual_Indicators2.19
			 );
		Valve26FB.In_Auto_SideA_Command:= FALSE;
		Valve26FB.In_Auto_SideB_Command:= FALSE;


	(*Valve 27, A+B*)
	(*spare*)
		Valve27FB
			(
			Enable_Motion:= Enable_Motion ,
			Enable_Latch:= TRUE,					(*Enabling Runs Valve as detent type (maintained solenoids*)
			Enable_SideA_PreCharge:= FALSE,		(*Enabling Turns Side A PreCharge Active, reset when Side B is energized in Auto*)
			Enable_SideB_PreCharge:= FALSE,		(*Enabling Turns Side B PreCharge Active, reset when Side A is energized in Auto*)
			PreCharge_Time:= T#0.10S,
			Enable_Auto_Commands:= In_Auto,
			Enable_Manual_Commands:= In_Manual AND All_Robots_Clear,
			In_Manual_SideA_Command:= Discrete_In.ManReqs2.20,
			In_Manual_SideB_Command:= Discrete_In.ManReqs2.21,
			SideA_Indicator:= FALSE,
			SideB_Indicator:= FALSE,
			TurnOn_SideA_SOL=> N101.Q.20,
			TurnOn_SideB_SOL=> N101.Q.21,
			TurnOn_SideA_Indicator=> Manual_Indicators2.20,
			TurnOn_SideB_Indicator=> Manual_Indicators2.21
			 );
		Valve27FB.In_Auto_SideA_Command:= FALSE;
		Valve27FB.In_Auto_SideB_Command:= FALSE;


	(*Valve 28, A+B*)
	(*spare*)
		Valve28FB
			(
			Enable_Motion:= Enable_Motion ,
			Enable_Latch:= TRUE,					(*Enabling Runs Valve as detent type (maintained solenoids*)
			Enable_SideA_PreCharge:= FALSE,		(*Enabling Turns Side A PreCharge Active, reset when Side B is energized in Auto*)
			Enable_SideB_PreCharge:= FALSE,		(*Enabling Turns Side B PreCharge Active, reset when Side A is energized in Auto*)
			PreCharge_Time:= T#0.10S,
			Enable_Auto_Commands:= In_Auto,
			Enable_Manual_Commands:= In_Manual AND All_Robots_Clear,
			In_Manual_SideA_Command:= Discrete_In.ManReqs2.22,
			In_Manual_SideB_Command:= Discrete_In.ManReqs2.23,
			SideA_Indicator:= FALSE,
			SideB_Indicator:= FALSE,
			TurnOn_SideA_SOL=> N101.Q.22,
			TurnOn_SideB_SOL=> N101.Q.23,
			TurnOn_SideA_Indicator=> Manual_Indicators2.22,
			TurnOn_SideB_Indicator=> Manual_Indicators2.23
			 );
		Valve28FB.In_Auto_SideA_Command:= FALSE;
		Valve28FB.In_Auto_SideB_Command:= FALSE;


	(*Valve 29, A+B*)
	(*spare*)
		Valve29FB
			(
			Enable_Motion:= Enable_Motion ,
			Enable_Latch:= TRUE,					(*Enabling Runs Valve as detent type (maintained solenoids*)
			Enable_SideA_PreCharge:= FALSE,		(*Enabling Turns Side A PreCharge Active, reset when Side B is energized in Auto*)
			Enable_SideB_PreCharge:= FALSE,		(*Enabling Turns Side B PreCharge Active, reset when Side A is energized in Auto*)
			PreCharge_Time:= T#0.10S,
			Enable_Auto_Commands:= In_Auto,
			Enable_Manual_Commands:= In_Manual AND All_Robots_Clear,
			In_Manual_SideA_Command:= Discrete_In.ManReqs2.24,
			In_Manual_SideB_Command:= Discrete_In.ManReqs2.25,
			SideA_Indicator:= FALSE,
			SideB_Indicator:= FALSE,
			TurnOn_SideA_SOL=> N101.Q.24,
			TurnOn_SideB_SOL=> N101.Q.25,
			TurnOn_SideA_Indicator=> Manual_Indicators2.24,
			TurnOn_SideB_Indicator=> Manual_Indicators2.25
			 );
		Valve29FB.In_Auto_SideA_Command:= FALSE;
		Valve29FB.In_Auto_SideB_Command:= FALSE;


	(*Valve 30, A+B*)
	(*spare*)
		Valve30FB
			(
			Enable_Motion:= Enable_Motion ,
			Enable_Latch:= TRUE,					(*Enabling Runs Valve as detent type (maintained solenoids*)
			Enable_SideA_PreCharge:= FALSE,		(*Enabling Turns Side A PreCharge Active, reset when Side B is energized in Auto*)
			Enable_SideB_PreCharge:= FALSE,		(*Enabling Turns Side B PreCharge Active, reset when Side A is energized in Auto*)
			PreCharge_Time:= T#0.10S,
			Enable_Auto_Commands:= In_Auto,
			Enable_Manual_Commands:= In_Manual AND All_Robots_Clear,
			In_Manual_SideA_Command:= Discrete_In.ManReqs2.26,
			In_Manual_SideB_Command:= Discrete_In.ManReqs2.27,
			SideA_Indicator:= FALSE,
			SideB_Indicator:= FALSE,
			TurnOn_SideA_SOL=> N101.Q.26,
			TurnOn_SideB_SOL=> N101.Q.27,
			TurnOn_SideA_Indicator=> Manual_Indicators2.26,
			TurnOn_SideB_Indicator=> Manual_Indicators2.27
			 );
		Valve30FB.In_Auto_SideA_Command:= FALSE;
		Valve30FB.In_Auto_SideB_Command:= FALSE;


	(*Valve 31, A+B*)
	(*spare*)
		Valve31FB
			(
			Enable_Motion:= Enable_Motion ,
			Enable_Latch:= TRUE,					(*Enabling Runs Valve as detent type (maintained solenoids*)
			Enable_SideA_PreCharge:= FALSE,		(*Enabling Turns Side A PreCharge Active, reset when Side B is energized in Auto*)
			Enable_SideB_PreCharge:= FALSE,		(*Enabling Turns Side B PreCharge Active, reset when Side A is energized in Auto*)
			PreCharge_Time:= T#0.10S,
			Enable_Auto_Commands:= In_Auto,
			Enable_Manual_Commands:= In_Manual AND All_Robots_Clear,
			In_Manual_SideA_Command:= Discrete_In.ManReqs2.28,
			In_Manual_SideB_Command:= Discrete_In.ManReqs2.29,
			SideA_Indicator:= FALSE,
			SideB_Indicator:= FALSE,
			TurnOn_SideA_SOL=> N101.Q.28,
			TurnOn_SideB_SOL=> N101.Q.29,
			TurnOn_SideA_Indicator=> Manual_Indicators2.28,
			TurnOn_SideB_Indicator=> Manual_Indicators2.29
			 );
		Valve31FB.In_Auto_SideA_Command:= FALSE;
		Valve31FB.In_Auto_SideB_Command:= FALSE;


	(*Valve 32, A+B*)
	(*spare*)
		Valve32FB
			(
			Enable_Motion:= Enable_Motion ,
			Enable_Latch:= TRUE,					(*Enabling Runs Valve as detent type (maintained solenoids*)
			Enable_SideA_PreCharge:= FALSE,		(*Enabling Turns Side A PreCharge Active, reset when Side B is energized in Auto*)
			Enable_SideB_PreCharge:= FALSE,		(*Enabling Turns Side B PreCharge Active, reset when Side A is energized in Auto*)
			PreCharge_Time:= T#0.10S,
			Enable_Auto_Commands:= In_Auto,
			Enable_Manual_Commands:= In_Manual AND All_Robots_Clear,
			In_Manual_SideA_Command:= Discrete_In.ManReqs2.30,
			In_Manual_SideB_Command:= Discrete_In.ManReqs2.31,
			SideA_Indicator:= FALSE,
			SideB_Indicator:= FALSE,
			TurnOn_SideA_SOL=> N101.Q.30,
			TurnOn_SideB_SOL=> N101.Q.31,
			TurnOn_SideA_Indicator=> Manual_Indicators2.30,
			TurnOn_SideB_Indicator=> Manual_Indicators2.31
			 );
		Valve32FB.In_Auto_SideA_Command:= FALSE;
		Valve32FB.In_Auto_SideB_Command:= FALSE;




















(*end*)
END_ACTION

ACTION ValveBank3:


(*+++++++++++THIS AREA IS CUSTOM PER INSTALLATION AND WILL HAVE TO BE MODIFIED PER +++++++++++++*)
(*+++++++++++THIS AREA IS CUSTOM PER INSTALLATION AND WILL HAVE TO BE MODIFIED PER +++++++++++++*)
(*+++++++++++THIS AREA IS CUSTOM PER INSTALLATION AND WILL HAVE TO BE MODIFIED PER +++++++++++++*)

(*+++++++++++VALVE BANK 3 +++++++++++++*)
(*+++++++++++VALVE BANK 3 +++++++++++++*)
(*+++++++++++VALVE BANK 3 +++++++++++++*)


	(*Valve 33, A+B*)
	(*spare*)
		Valve33FB
			(
			Enable_Motion:= Enable_Motion ,
			Enable_Latch:= TRUE,					(*Enabling Runs Valve as detent type (maintained solenoids*)
			Enable_SideA_PreCharge:= FALSE,		(*Enabling Turns Side A PreCharge Active, reset when Side B is energized in Auto*)
			Enable_SideB_PreCharge:= FALSE,		(*Enabling Turns Side B PreCharge Active, reset when Side A is energized in Auto*)
			PreCharge_Time:= T#0.1S,
			Enable_Auto_Commands:= In_Auto,
			Enable_Manual_Commands:= In_Manual AND All_Robots_Clear,
			In_Manual_SideA_Command:= Discrete_In.ManReqs3.0,
			In_Manual_SideB_Command:= (Discrete_In.ManReqs3.1 OR Discrete_In.Go_Home),
			SideA_Indicator:= FALSE,
			SideB_Indicator:= FALSE,
			TurnOn_SideA_SOL=> N102.Q.0,
			TurnOn_SideB_SOL=> N102.Q.1,
			TurnOn_SideA_Indicator=> Manual_Indicators3.0,
			TurnOn_SideB_Indicator=> Manual_Indicators3.1
			 );
		Valve33FB.In_Auto_SideA_Command:= FALSE;
		Valve33FB.In_Auto_SideB_Command:= FALSE;


	(*Valve 34, A+B*)
	(*spare*)
		Valve34FB
			(
			Enable_Motion:= Enable_Motion ,
			Enable_Latch:= TRUE,					(*Enabling Runs Valve as detent type (maintained solenoids*)
			Enable_SideA_PreCharge:= FALSE,		(*Enabling Turns Side A PreCharge Active, reset when Side B is energized in Auto*)
			Enable_SideB_PreCharge:= FALSE,		(*Enabling Turns Side B PreCharge Active, reset when Side A is energized in Auto*)
			PreCharge_Time:= T#0.10S,
			Enable_Auto_Commands:= In_Auto,
			Enable_Manual_Commands:= In_Manual AND All_Robots_Clear,
			In_Manual_SideA_Command:= Discrete_In.ManReqs3.2,
			In_Manual_SideB_Command:= Discrete_In.ManReqs3.3,
			SideA_Indicator:= FALSE,
			SideB_Indicator:= FALSE,
			TurnOn_SideA_SOL=> N102.Q.2,
			TurnOn_SideB_SOL=> N102.Q.3,
			TurnOn_SideA_Indicator=> Manual_Indicators3.2,
			TurnOn_SideB_Indicator=> Manual_Indicators3.3
			 );
		Valve34FB.In_Auto_SideA_Command:= FALSE;
		Valve34FB.In_Auto_SideB_Command:= FALSE;


	(*Valve 35, A+B*)
	(*spare*)
		Valve35FB
			(
			Enable_Motion:= Enable_Motion ,
			Enable_Latch:= TRUE,					(*Enabling Runs Valve as detent type (maintained solenoids*)
			Enable_SideA_PreCharge:= FALSE,		(*Enabling Turns Side A PreCharge Active, reset when Side B is energized in Auto*)
			Enable_SideB_PreCharge:= FALSE,		(*Enabling Turns Side B PreCharge Active, reset when Side A is energized in Auto*)
			PreCharge_Time:= T#0.10S,
			Enable_Auto_Commands:= In_Auto,
			Enable_Manual_Commands:= In_Manual AND All_Robots_Clear,
			In_Manual_SideA_Command:= Discrete_In.ManReqs3.4,
			In_Manual_SideB_Command:= Discrete_In.ManReqs3.5,
			SideA_Indicator:= FALSE,
			SideB_Indicator:= FALSE,
			TurnOn_SideA_SOL=> N102.Q.4,
			TurnOn_SideB_SOL=> N102.Q.5,
			TurnOn_SideA_Indicator=> Manual_Indicators3.4,
			TurnOn_SideB_Indicator=> Manual_Indicators3.5
			 );
		Valve35FB.In_Auto_SideA_Command:= FALSE;
		Valve35FB.In_Auto_SideB_Command:= FALSE;


	(*Valve 36, A+B*)
	(*spare*)
		Valve36FB
			(
			Enable_Motion:= Enable_Motion ,
			Enable_Latch:= TRUE,					(*Enabling Runs Valve as detent type (maintained solenoids*)
			Enable_SideA_PreCharge:= FALSE,		(*Enabling Turns Side A PreCharge Active, reset when Side B is energized in Auto*)
			Enable_SideB_PreCharge:= FALSE,		(*Enabling Turns Side B PreCharge Active, reset when Side A is energized in Auto*)
			PreCharge_Time:= T#0.10S,
			Enable_Auto_Commands:= In_Auto,
			Enable_Manual_Commands:= In_Manual AND All_Robots_Clear,
			In_Manual_SideA_Command:= Discrete_In.ManReqs3.6,
			In_Manual_SideB_Command:= Discrete_In.ManReqs3.7,
			SideA_Indicator:= FALSE,
			SideB_Indicator:= FALSE,
			TurnOn_SideA_SOL=> N102.Q.6,
			TurnOn_SideB_SOL=> N102.Q.7,
			TurnOn_SideA_Indicator=> Manual_Indicators3.6,
			TurnOn_SideB_Indicator=> Manual_Indicators3.7
			 );
		Valve36FB.In_Auto_SideA_Command:= FALSE;
		Valve36FB.In_Auto_SideB_Command:= FALSE;


	(*Valve 37, A+B*)
	(*spare*)
		Valve37FB
			(
			Enable_Motion:= Enable_Motion ,
			Enable_Latch:= TRUE,					(*Enabling Runs Valve as detent type (maintained solenoids*)
			Enable_SideA_PreCharge:= FALSE,		(*Enabling Turns Side A PreCharge Active, reset when Side B is energized in Auto*)
			Enable_SideB_PreCharge:= FALSE,		(*Enabling Turns Side B PreCharge Active, reset when Side A is energized in Auto*)
			PreCharge_Time:= T#0.10S,
			Enable_Auto_Commands:= In_Auto,
			Enable_Manual_Commands:= In_Manual AND All_Robots_Clear,
			In_Manual_SideA_Command:= Discrete_In.ManReqs3.8,
			In_Manual_SideB_Command:= Discrete_In.ManReqs3.9,
			SideA_Indicator:= FALSE,
			SideB_Indicator:= FALSE,
			TurnOn_SideA_SOL=> N102.Q.8,
			TurnOn_SideB_SOL=> N102.Q.9,
			TurnOn_SideA_Indicator=> Manual_Indicators3.8,
			TurnOn_SideB_Indicator=> Manual_Indicators3.9
			 );
		Valve37FB.In_Auto_SideA_Command:= FALSE;
		Valve37FB.In_Auto_SideB_Command:= FALSE;


	(*Valve 38, A+B*)
	(*spare*)
		Valve38FB
			(
			Enable_Motion:= Enable_Motion ,
			Enable_Latch:= TRUE,					(*Enabling Runs Valve as detent type (maintained solenoids*)
			Enable_SideA_PreCharge:= FALSE,		(*Enabling Turns Side A PreCharge Active, reset when Side B is energized in Auto*)
			Enable_SideB_PreCharge:= FALSE,		(*Enabling Turns Side B PreCharge Active, reset when Side A is energized in Auto*)
			PreCharge_Time:= T#0.10S,
			Enable_Auto_Commands:= In_Auto,
			Enable_Manual_Commands:= In_Manual AND All_Robots_Clear,
			In_Manual_SideA_Command:= Discrete_In.ManReqs3.10,
			In_Manual_SideB_Command:= Discrete_In.ManReqs3.11,
			SideA_Indicator:= FALSE,
			SideB_Indicator:= FALSE,
			TurnOn_SideA_SOL=> N102.Q.10,
			TurnOn_SideB_SOL=> N102.Q.11,
			TurnOn_SideA_Indicator=> Manual_Indicators3.10,
			TurnOn_SideB_Indicator=> Manual_Indicators3.11
			 );
		Valve38FB.In_Auto_SideA_Command:= FALSE;
		Valve38FB.In_Auto_SideB_Command:= FALSE;


	(*Valve 39, A+B*)
	(*spare*)
		Valve39FB
			(
			Enable_Motion:= Enable_Motion ,
			Enable_Latch:= TRUE,					(*Enabling Runs Valve as detent type (maintained solenoids*)
			Enable_SideA_PreCharge:= FALSE,		(*Enabling Turns Side A PreCharge Active, reset when Side B is energized in Auto*)
			Enable_SideB_PreCharge:= FALSE,		(*Enabling Turns Side B PreCharge Active, reset when Side A is energized in Auto*)
			PreCharge_Time:= T#0.10S,
			Enable_Auto_Commands:= In_Auto,
			Enable_Manual_Commands:= In_Manual AND All_Robots_Clear,
			In_Manual_SideA_Command:= Discrete_In.ManReqs3.12,
			In_Manual_SideB_Command:= Discrete_In.ManReqs3.13,
			SideA_Indicator:= FALSE,
			SideB_Indicator:= FALSE,
			TurnOn_SideA_SOL=> N102.Q.12,
			TurnOn_SideB_SOL=> N102.Q.13,
			TurnOn_SideA_Indicator=> Manual_Indicators3.12,
			TurnOn_SideB_Indicator=> Manual_Indicators3.13
			 );
		Valve39FB.In_Auto_SideA_Command:= FALSE;
		Valve39FB.In_Auto_SideB_Command:= FALSE;


	(*Valve 40, A+B*)
	(*spare*)
		Valve40FB
			(
			Enable_Motion:= Enable_Motion ,
			Enable_Latch:= TRUE,					(*Enabling Runs Valve as detent type (maintained solenoids*)
			Enable_SideA_PreCharge:= FALSE,		(*Enabling Turns Side A PreCharge Active, reset when Side B is energized in Auto*)
			Enable_SideB_PreCharge:= FALSE,		(*Enabling Turns Side B PreCharge Active, reset when Side A is energized in Auto*)
			PreCharge_Time:= T#0.10S,
			Enable_Auto_Commands:= In_Auto,
			Enable_Manual_Commands:= In_Manual AND All_Robots_Clear,
			In_Manual_SideA_Command:= Discrete_In.ManReqs3.14,
			In_Manual_SideB_Command:= Discrete_In.ManReqs3.15,
			SideA_Indicator:= FALSE,
			SideB_Indicator:= FALSE,
			TurnOn_SideA_SOL=> N102.Q.14,
			TurnOn_SideB_SOL=> N102.Q.15,
			TurnOn_SideA_Indicator=> Manual_Indicators3.14,
			TurnOn_SideB_Indicator=> Manual_Indicators3.15
			 );
		Valve40FB.In_Auto_SideA_Command:= FALSE;
		Valve40FB.In_Auto_SideB_Command:= FALSE;


	(*Valve 41, A+B*)
	(*spare*)
		Valve41FB
			(
			Enable_Motion:= Enable_Motion ,
			Enable_Latch:= TRUE,					(*Enabling Runs Valve as detent type (maintained solenoids*)
			Enable_SideA_PreCharge:= FALSE,		(*Enabling Turns Side A PreCharge Active, reset when Side B is energized in Auto*)
			Enable_SideB_PreCharge:= FALSE,		(*Enabling Turns Side B PreCharge Active, reset when Side A is energized in Auto*)
			PreCharge_Time:= T#0.10S,
			Enable_Auto_Commands:= In_Auto,
			Enable_Manual_Commands:= In_Manual AND All_Robots_Clear,
			In_Manual_SideA_Command:= Discrete_In.ManReqs3.16,
			In_Manual_SideB_Command:= Discrete_In.ManReqs3.17,
			SideA_Indicator:= FALSE,
			SideB_Indicator:= FALSE,
			TurnOn_SideA_SOL=> N102.Q.16,
			TurnOn_SideB_SOL=> N102.Q.17,
			TurnOn_SideA_Indicator=> Manual_Indicators3.16,
			TurnOn_SideB_Indicator=> Manual_Indicators3.17
			 );
		Valve41FB.In_Auto_SideA_Command:= FALSE;
		Valve41FB.In_Auto_SideB_Command:= FALSE;


	(*Valve 42, A+B*)
	(*spare*)
		Valve42FB
			(
			Enable_Motion:= Enable_Motion ,
			Enable_Latch:= TRUE,					(*Enabling Runs Valve as detent type (maintained solenoids*)
			Enable_SideA_PreCharge:= FALSE,		(*Enabling Turns Side A PreCharge Active, reset when Side B is energized in Auto*)
			Enable_SideB_PreCharge:= FALSE,		(*Enabling Turns Side B PreCharge Active, reset when Side A is energized in Auto*)
			PreCharge_Time:= T#0.10S,
			Enable_Auto_Commands:= In_Auto,
			Enable_Manual_Commands:= In_Manual AND All_Robots_Clear,
			In_Manual_SideA_Command:= Discrete_In.ManReqs3.18,
			In_Manual_SideB_Command:= Discrete_In.ManReqs3.19,
			SideA_Indicator:= FALSE,
			SideB_Indicator:= FALSE,
			TurnOn_SideA_SOL=> N102.Q.18,
			TurnOn_SideB_SOL=> N102.Q.19,
			TurnOn_SideA_Indicator=> Manual_Indicators3.18,
			TurnOn_SideB_Indicator=> Manual_Indicators3.19
			 );
		Valve42FB.In_Auto_SideA_Command:= FALSE;
		Valve42FB.In_Auto_SideB_Command:= FALSE;


	(*Valve 43, A+B*)
	(*spare*)
		Valve43FB
			(
			Enable_Motion:= Enable_Motion ,
			Enable_Latch:= TRUE,					(*Enabling Runs Valve as detent type (maintained solenoids*)
			Enable_SideA_PreCharge:= FALSE,		(*Enabling Turns Side A PreCharge Active, reset when Side B is energized in Auto*)
			Enable_SideB_PreCharge:= FALSE,		(*Enabling Turns Side B PreCharge Active, reset when Side A is energized in Auto*)
			PreCharge_Time:= T#0.10S,
			Enable_Auto_Commands:= In_Auto,
			Enable_Manual_Commands:= In_Manual AND All_Robots_Clear,
			In_Manual_SideA_Command:= Discrete_In.ManReqs3.20,
			In_Manual_SideB_Command:= Discrete_In.ManReqs3.21,
			SideA_Indicator:= FALSE,
			SideB_Indicator:= FALSE,
			TurnOn_SideA_SOL=> N102.Q.20,
			TurnOn_SideB_SOL=> N102.Q.21,
			TurnOn_SideA_Indicator=> Manual_Indicators3.20,
			TurnOn_SideB_Indicator=> Manual_Indicators3.21
			 );
		Valve43FB.In_Auto_SideA_Command:= FALSE;
		Valve43FB.In_Auto_SideB_Command:= FALSE;


	(*Valve 44, A+B*)
	(*spare*)
		Valve44FB
			(
			Enable_Motion:= Enable_Motion ,
			Enable_Latch:= TRUE,					(*Enabling Runs Valve as detent type (maintained solenoids*)
			Enable_SideA_PreCharge:= FALSE,		(*Enabling Turns Side A PreCharge Active, reset when Side B is energized in Auto*)
			Enable_SideB_PreCharge:= FALSE,		(*Enabling Turns Side B PreCharge Active, reset when Side A is energized in Auto*)
			PreCharge_Time:= T#0.10S,
			Enable_Auto_Commands:= In_Auto,
			Enable_Manual_Commands:= In_Manual AND All_Robots_Clear,
			In_Manual_SideA_Command:= Discrete_In.ManReqs3.22,
			In_Manual_SideB_Command:= Discrete_In.ManReqs3.23,
			SideA_Indicator:= FALSE,
			SideB_Indicator:= FALSE,
			TurnOn_SideA_SOL=> N102.Q.22,
			TurnOn_SideB_SOL=> N102.Q.23,
			TurnOn_SideA_Indicator=> Manual_Indicators3.22,
			TurnOn_SideB_Indicator=> Manual_Indicators3.23
			 );
		Valve44FB.In_Auto_SideA_Command:= FALSE;
		Valve44FB.In_Auto_SideB_Command:= FALSE;


	(*Valve 45, A+B*)
	(*spare*)
		Valve45FB
			(
			Enable_Motion:= Enable_Motion ,
			Enable_Latch:= TRUE,					(*Enabling Runs Valve as detent type (maintained solenoids*)
			Enable_SideA_PreCharge:= FALSE,		(*Enabling Turns Side A PreCharge Active, reset when Side B is energized in Auto*)
			Enable_SideB_PreCharge:= FALSE,		(*Enabling Turns Side B PreCharge Active, reset when Side A is energized in Auto*)
			PreCharge_Time:= T#0.10S,
			Enable_Auto_Commands:= In_Auto,
			Enable_Manual_Commands:= In_Manual AND All_Robots_Clear,
			In_Manual_SideA_Command:= Discrete_In.ManReqs3.24,
			In_Manual_SideB_Command:= Discrete_In.ManReqs3.25,
			SideA_Indicator:= FALSE,
			SideB_Indicator:= FALSE,
			TurnOn_SideA_SOL=> N102.Q.24,
			TurnOn_SideB_SOL=> N102.Q.25,
			TurnOn_SideA_Indicator=> Manual_Indicators3.24,
			TurnOn_SideB_Indicator=> Manual_Indicators3.25
			 );
		Valve45FB.In_Auto_SideA_Command:= FALSE;
		Valve45FB.In_Auto_SideB_Command:= FALSE;


	(*Valve 46, A+B*)
	(*spare*)
		Valve46FB
			(
			Enable_Motion:= Enable_Motion ,
			Enable_Latch:= TRUE,					(*Enabling Runs Valve as detent type (maintained solenoids*)
			Enable_SideA_PreCharge:= FALSE,		(*Enabling Turns Side A PreCharge Active, reset when Side B is energized in Auto*)
			Enable_SideB_PreCharge:= FALSE,		(*Enabling Turns Side B PreCharge Active, reset when Side A is energized in Auto*)
			PreCharge_Time:= T#0.10S,
			Enable_Auto_Commands:= In_Auto,
			Enable_Manual_Commands:= In_Manual AND All_Robots_Clear,
			In_Manual_SideA_Command:= Discrete_In.ManReqs3.26,
			In_Manual_SideB_Command:= Discrete_In.ManReqs3.27,
			SideA_Indicator:= FALSE,
			SideB_Indicator:= FALSE,
			TurnOn_SideA_SOL=> N102.Q.26,
			TurnOn_SideB_SOL=> N102.Q.27,
			TurnOn_SideA_Indicator=> Manual_Indicators3.26,
			TurnOn_SideB_Indicator=> Manual_Indicators3.27
			 );
		Valve46FB.In_Auto_SideA_Command:= FALSE;
		Valve46FB.In_Auto_SideB_Command:= FALSE;


	(*Valve 47, A+B*)
	(*spare*)
		Valve47FB
			(
			Enable_Motion:= Enable_Motion ,
			Enable_Latch:= TRUE,					(*Enabling Runs Valve as detent type (maintained solenoids*)
			Enable_SideA_PreCharge:= FALSE,		(*Enabling Turns Side A PreCharge Active, reset when Side B is energized in Auto*)
			Enable_SideB_PreCharge:= FALSE,		(*Enabling Turns Side B PreCharge Active, reset when Side A is energized in Auto*)
			PreCharge_Time:= T#0.10S,
			Enable_Auto_Commands:= In_Auto,
			Enable_Manual_Commands:= In_Manual AND All_Robots_Clear,
			In_Manual_SideA_Command:= Discrete_In.ManReqs3.28,
			In_Manual_SideB_Command:= Discrete_In.ManReqs3.29,
			SideA_Indicator:= FALSE,
			SideB_Indicator:= FALSE,
			TurnOn_SideA_SOL=> N102.Q.28,
			TurnOn_SideB_SOL=> N102.Q.29,
			TurnOn_SideA_Indicator=> Manual_Indicators3.28,
			TurnOn_SideB_Indicator=> Manual_Indicators3.29
			 );
		Valve47FB.In_Auto_SideA_Command:= FALSE;
		Valve47FB.In_Auto_SideB_Command:= FALSE;


	(*Valve 48, A+B*)
	(*spare*)
		Valve48FB
			(
			Enable_Motion:= Enable_Motion ,
			Enable_Latch:= TRUE,					(*Enabling Runs Valve as detent type (maintained solenoids*)
			Enable_SideA_PreCharge:= FALSE,		(*Enabling Turns Side A PreCharge Active, reset when Side B is energized in Auto*)
			Enable_SideB_PreCharge:= FALSE,		(*Enabling Turns Side B PreCharge Active, reset when Side A is energized in Auto*)
			PreCharge_Time:= T#0.10S,
			Enable_Auto_Commands:= In_Auto,
			Enable_Manual_Commands:= In_Manual AND All_Robots_Clear,
			In_Manual_SideA_Command:= Discrete_In.ManReqs3.30,
			In_Manual_SideB_Command:= Discrete_In.ManReqs3.31,
			SideA_Indicator:= FALSE,
			SideB_Indicator:= FALSE,
			TurnOn_SideA_SOL=> N102.Q.30,
			TurnOn_SideB_SOL=> N102.Q.31,
			TurnOn_SideA_Indicator=> Manual_Indicators3.30,
			TurnOn_SideB_Indicator=> Manual_Indicators3.31
			 );
		Valve48FB.In_Auto_SideA_Command:= FALSE;
		Valve48FB.In_Auto_SideB_Command:= FALSE;


























(*end*)
END_ACTION

ACTION Xfer_To_UI:
(*Transfer General Status of Fixture and I/O Images for Display On HMI*)
	Discrete_Image.Status:= Status;
	Discrete_Image.CLFaults1:= CLFaults1;
	Discrete_Image.CLFaults2:= CLFaults2;
	Discrete_Image.CLFaults3:= CLFaults3;
	Discrete_Image.CLFaults4:= CLFaults4;
	Discrete_Image.CLFaulted:= CLFaulted;
	Discrete_Image.PPFaults:= PPFaults;
	Discrete_Image.PPFaults1:= PPFaults1;
	Discrete_Image.PPFaults2:= PPFaults2;
	Discrete_Image.PPFaulted:= PPFaulted;
	Discrete_Image.Model_Data:= Model_ID;
	Discrete_Image.ToolID:= Fix_ID;
	Discrete_Image.ProdCount:= Prod_Count_Out;
	Discrete_Image.CycleTime:= Cycle_Time_Out;
	Discrete_Image.PrevCycleTime:= PrevCycle_Time_Out;
	Discrete_Image.LoadTime:= Load_Time_Out;
	Discrete_Image.WeldTime:= Weld_Time_Out;
	Discrete_Image.UnloadTime:= Unload_Time_Out;

	Discrete_Image.InAuto:= In_Auto_Mode;
	Discrete_Image.InManual:= In_Manual_Mode;
	Discrete_Image.ManInds:= Manual_Indicators1;
	Discrete_Image.ManInds2:= Manual_Indicators2;
	Discrete_Image.ManInds3:= Manual_Indicators3;
	Discrete_Image.At_Home:= Tool_At_Home;
	Discrete_Image.Enable_Motion:= Enable_Motion;
	Discrete_Image.All_Sensors_Off:= All_Sensors_Off;
	Discrete_Image.Bypass_ACKS:= Discrete_In.Bypass_REQS;
	Discrete_Image.CustomApplication_ACKS:= Discrete_In.CustomApplication_REQS;
	Discrete_Image.Fixture_Allow_Model_Change:= Fixture_Allow_Model_Change;
	Discrete_Image.NodeLayout:=NodeLayout;
	Discrete_Image.NodeState:=NodeState;
	
	Discrete_Image.Input_Node_Count:= Discrete_In.Input_Node_Count;
	Discrete_Image.VB_Node_Count:= Discrete_In.VB_Node_Count;
	Discrete_Image.Water_Stand_Count:= Discrete_In.Water_Stand_Count;

	IF  (Discrete_Image.Input_Node_Count < 4)
		THEN Discrete_Image.VB_Screen_Position:= 1;
	ELSIF  (Discrete_Image.Input_Node_Count < 7)
		THEN Discrete_Image.VB_Screen_Position:= 2;
	ELSIF  (Discrete_Image.Input_Node_Count < 10)
		THEN Discrete_Image.VB_Screen_Position:= 3;
	ELSIF  (Discrete_Image.Input_Node_Count < 13)
		THEN Discrete_Image.VB_Screen_Position:= 4;
	ELSIF  (Discrete_Image.Input_Node_Count < 16)
		THEN Discrete_Image.VB_Screen_Position:= 5;
	ELSIF  (Discrete_Image.Input_Node_Count < 19)
		THEN Discrete_Image.VB_Screen_Position:= 6;
	ELSIF  (Discrete_Image.Input_Node_Count < 22)
		THEN Discrete_Image.VB_Screen_Position:= 7;
	ELSIF  (Discrete_Image.Input_Node_Count < 26)
		THEN Discrete_Image.VB_Screen_Position:= 8;
	ELSE
			Discrete_Image.VB_Screen_Position:= 9;
	END_IF;

	Discrete_Image.N00:= N00;
	Discrete_Image.N01:= N01;
	Discrete_Image.N02:= N02;
	Discrete_Image.N03:= N03;
	Discrete_Image.N04:= N04;
	Discrete_Image.N05:= N05;
	Discrete_Image.N06:= N06;
	Discrete_Image.N07:= N07;
	Discrete_Image.N08:= N08;
	Discrete_Image.N09:= N09;
	Discrete_Image.N10:= N10;
	Discrete_Image.N11:= N11;
	Discrete_Image.N12:= N12;
	Discrete_Image.N13:= N13;
	Discrete_Image.N14:= N14;
	Discrete_Image.N15:= N15;
	Discrete_Image.N16:= N16;
	Discrete_Image.N17:= N17;
	Discrete_Image.N18:= N18;
	Discrete_Image.N19:= N19;
	Discrete_Image.N20:= N20;
	Discrete_Image.N21:= N21;
	Discrete_Image.N22:= N22;
	Discrete_Image.N100:= N100;
	Discrete_Image.N100_STAT:= N100_STAT;
	Discrete_Image.N101:= N101;
	Discrete_Image.N101_STAT:= N101_STAT;
	Discrete_Image.N102:= N102;
	Discrete_Image.N102_STAT:= N102_STAT;
	
	(*IsEnabled control For UI screen: Default "IsEnabled == True"*)
	Discrete_Image.Enable_FixtureContext_Clamps:= TRUE;
	Discrete_Image.Enable_FixtureContext_QA:= TRUE;
	Discrete_Image.Enable_FixtureContext_Manual:= TRUE;


	Discrete_Image.ECatSlave_Cable_Breaks:= ECatSlave_Cable_Breaks;

	Discrete_Image.Operator_Performance_Pen:= Production_Report.Shift_Report[0].Prod_Performance;
END_ACTION

END_PROGRAM

// ---- POUs/Fixtures and EOAT/Human/Fix04.TcPOU
(*Fixture*)

PROGRAM Fix04
	VAR_INPUT
		Enable_Prog: BOOL;
		Enable_Motion: BOOL;
		Discrete_In: udt_FixXX_Input_Image_20180202;
		Dry_Cycle: BOOL;
		Cell_In_Services: BOOL;
		Flash_Rate: BOOL;
		NodeLayout:udt_ECATNodeData_20221507;

	END_VAR

	VAR
(*Hardware Related Data Types*)
			(*Develop "Beckhoff Nodes"*)
			{attribute 'OPC.UA.DA':='1'}
			N00 AT %I*: udt_EP1111;
			{attribute 'OPC.UA.DA':='1'}
			N01 AT %I*: udt_EP1008_002_v2;
			{attribute 'OPC.UA.DA':='1'}
			N02 AT %I*: udt_EP1008_002_v2;
			{attribute 'OPC.UA.DA':='1'}
			N03 AT %I*: udt_EP1008_002_v2;
			{attribute 'OPC.UA.DA':='1'}
			N04 AT %I*: udt_EP1008_002_v2;
			{attribute 'OPC.UA.DA':='1'}
			N05 AT %I*: udt_EP1008_002_v2;
			{attribute 'OPC.UA.DA':='1'}
			N06 AT %I*: udt_EP1008_002_v2;
			{attribute 'OPC.UA.DA':='1'}
			N07 AT %I*: udt_EP1008_002_v2;
			{attribute 'OPC.UA.DA':='1'}
			N08 AT %I*: udt_EP1008_002_v2;
			{attribute 'OPC.UA.DA':='1'}
			N09 AT %I*: udt_EP1008_002_v2;
			{attribute 'OPC.UA.DA':='1'}
			N10 AT %I*: udt_EP1008_002_v2;
			{attribute 'OPC.UA.DA':='1'}
			N11 AT %I*: udt_EP1008_002_v2;
			{attribute 'OPC.UA.DA':='1'}
			N12 AT %I*: udt_EP1008_002_v2;
			{attribute 'OPC.UA.DA':='1'}
			N13 AT %I*: udt_EP1008_002_v2;
			{attribute 'OPC.UA.DA':='1'}
			N14 AT %I*: udt_EP1008_002_v2;
			{attribute 'OPC.UA.DA':='1'}
			N15 AT %I*: udt_EP1008_002_v2;
			{attribute 'OPC.UA.DA':='1'}
			N16 AT %I*: udt_EP1008_002_v2;
			{attribute 'OPC.UA.DA':='1'}
			N17 AT %I*: udt_EP1008_002_v2;
			{attribute 'OPC.UA.DA':='1'}
			N18 AT %I*: udt_EP1008_002_v2;
			{attribute 'OPC.UA.DA':='1'}
			N19 AT %I*: udt_EP1008_002_v2;
			{attribute 'OPC.UA.DA':='1'}
			N20 AT %I*: udt_EP1008_002_v2;
			{attribute 'OPC.UA.DA':='1'}
			N21 AT %I*: udt_EP1008_002_v2;
			{attribute 'OPC.UA.DA':='1'}
			N22 AT %I*: udt_EP1008_002_v2;
			{attribute 'OPC.UA.DA':='1'}
			N100 AT %Q*: udt_SMC_EX260_ValveBank;
			{attribute 'OPC.UA.DA':='1'}
			N100_STAT AT %I*:udt_SMC_EX260_Stat;
			{attribute 'OPC.UA.DA':='1'}
			N101 AT %Q*: udt_SMC_EX260_ValveBank;
			{attribute 'OPC.UA.DA':='1'}
			N101_STAT AT %I*:udt_SMC_EX260_Stat;
			{attribute 'OPC.UA.DA':='1'}
			N102 AT %Q*: udt_SMC_EX260_ValveBank;
			{attribute 'OPC.UA.DA':='1'}
			N102_STAT AT %I*:udt_SMC_EX260_Stat;
			
			
			(*Added nodes - AB*)
			N90_STAT AT %I*: udt_EP9214_STAT_20250704;
			N90_CMD AT %Q*: udt_EP9214_CMD_20250704;
			N98 : udt_EP2328_0002;

(* Nodes States*)
		NodeState: ARRAY[0..63] OF UINT;
		DiscreteNode_OK: BOOL;
(*Cable Break States*)
		ECatSlave_Cable_Breaks: ARRAY[0..1] OF DINT;
(*Standard Internal Variables*)
		(*Generic Sensor Variables*)
		All_Sensors_On: UINT;
		All_Sensors_Off: BOOL;
		All_Sensors_Off1: BOOL;
		All_Sensors_Off2: BOOL;
		(*Generic Position Variables*)
		Tool_At_Home: BOOL;
		Tool_At_Load: UINT;
		Tool_At_Weld: UINT;
		Tool_At_Rotate: UINT;
		Tool_At_Seal: UINT;
		Tool_At_Stud: UINT;
		Tool_At_Unload: UINT ;
		(*Grouping Of Items*)
		All_QAChecks_OK: BOOL;
		QAChecks_Failed: BOOL;
		(*General Internals*)
		In_Auto: BOOL;
		In_Manual: BOOL;

		Auto_Run: BOOL;
		Reset_All_Completes:BOOL;
		Load_Robots_Clear1: BOOL;
		Load_Robots_Clear2: BOOL;
		Load_Robots_Clear: BOOL;
		Load_Robots_WorkingOK1: BOOL;
		Load_Robots_WorkingOK2: BOOL;
		Load_Robots_Complete1: BOOL;
		Load_Robots_Complete2: BOOL;
		Load_Robots_PartInEOAT1: BOOL;
		Load_Robots_PartInEOAT2: BOOL;
		Load_Robots_UnclampEarly1: BOOL;
		Load_Robots_UnclampEarly2: BOOL;
		Seal_Robots_Clear: BOOL;
		Seal_Robots_WorkingOK: BOOL;
		Seal_Robots_UnclampEarly: BOOL;
		Seal_Robots_Complete: BOOL;
		Stud_Robots_Clear: BOOL;
		Stud_Robots_WorkingOK: BOOL;
		Stud_Robots_UnclampEarly: BOOL;
		Stud_Robots_Complete: BOOL;
		Weld_Robots_Clear: BOOL;
		Weld_Robots_WorkingOK: BOOL;
		Weld_Robots_UnclampEarly: BOOL;
		Weld_Robots_Complete: BOOL;
		Mig_Robots_Ready :BOOL;
		TurntableA_Clear: BOOL;
		TurntableB_Clear: BOOL;
		Turntable_Clear:BOOL;
		Turntable_WorkingOK: BOOL;
		TurntableA_Complete: BOOL;
		TurntableB_Complete: BOOL;
		Unload_Robots_Clear1: BOOL;
		Unload_Robots_WorkingOK1: BOOL;
		Unload_Robots_Complete1: BOOL;
		Unload_Robots_EOATEmpty1: BOOL;
		Unload_Robots_Clear2: BOOL;
		Unload_Robots_WorkingOK2: BOOL;
		Unload_Robots_Complete2: BOOL;
		Unload_Robots_EOATEmpty2: BOOL;
		Unload_Robots_Clear: BOOL;
		All_Robots_Clear: BOOL;

		Unload_Robot_Complete: BOOL;

		Start_Load_Robots1: BOOL;
		Start_Load_Robots2: BOOL;
		Start_Weld_Robots: BOOL;
		Start_Unload_Robots1: BOOL;
		Start_Unload_Robots2: BOOL;
		Start_Seal_Robots: BOOL;
		Start_Stud_Robots: BOOL;
		Start_TurntableA: BOOL;
		Start_TurntableB: BOOL;
		Load_Robots_Proceed1: BOOL;
		Load_Robots_Proceed2: BOOL;
		Weld_Robots_Proceed: BOOL;
		Seal_Robots_Proceed: BOOL;
		Stud_Robots_Proceed: BOOL;
		Unload_Robots_Proceed1: BOOL;
		Unload_Robots_Proceed2: BOOL;

		Prod_Inc: R_TRIG;
		Cycle_Time: TON;
		Cycle_Time_Pulse: R_TRIG;
		Load_Time: TON;
		Weld_Time: TON;
		Seal_Time: TON;
		Stud_Time: TON;
		Turn_Time: TON;
		Unload_Time: TON;
		Date_Stamp_TMR: TON;
		Date_StampHome_TMR: TON;
		CLFaulted: UDINT;
		PPFaulted: UDINT;
		Manual_Ind_HomePrompt: BOOL;
		Fixture_Allow_Model_Change: BOOL;

(*Non-Standard Variables*)

		(*FB Instances*)
		Clamp1FB: FB_Cylinder_Status;
		Clamp2FB: FB_Cylinder_Status;
		Clamp3FB: FB_Cylinder_Status;
		Clamp4FB: FB_Cylinder_Status;
		Clamp5FB: FB_Cylinder_Status;
		Clamp6FB: FB_Cylinder_Status;
		Clamp7FB: FB_Cylinder_Status;
		Clamp8FB: FB_Cylinder_Status;
		Clamp9FB: FB_Cylinder_Status;
		Clamp10FB: FB_Cylinder_Status;
		Clamp11FB: FB_Cylinder_Status;
		Clamp12FB: FB_Cylinder_Status;
		Clamp13FB: FB_Cylinder_Status;
		Clamp14FB: FB_Cylinder_Status;
		Clamp15FB: FB_Cylinder_Status;
		Clamp16FB: FB_Cylinder_Status;
		Clamp17FB: FB_Cylinder_Status;
		Clamp18FB: FB_Cylinder_Status;
		Clamp19FB: FB_Cylinder_Status;
		Clamp20FB: FB_Cylinder_Status;
		Clamp21FB: FB_Cylinder_Status;
		Clamp22FB: FB_Cylinder_Status;
		Clamp23FB: FB_Cylinder_Status;
		Clamp24FB: FB_Cylinder_Status;
		Cyl1FB: FB_TripleCylinder_20150625;
		Pin1FB: FB_Cylinder_Status;
		Pin2FB: FB_Cylinder_Status;
		Pin3FB: FB_Cylinder_Status;
		Pin4FB: FB_Cylinder_Status;
		Pin5FB: FB_Cylinder_Status;
		Pin6FB: FB_Cylinder_Status;
		Pin7FB: FB_Cylinder_Status;
		Pin8FB: FB_Cylinder_Status;
		Pin9FB: FB_Cylinder_Status;
		Pin10FB: FB_Cylinder_Status;
		Pin11FB: FB_Cylinder_Status;
		Pin12FB: FB_Cylinder_Status;
		Pin13FB: FB_Cylinder_Status;
		Pin14FB: FB_Cylinder_Status;
		Pin15FB: FB_Cylinder_Status;
		Pin16FB: FB_Cylinder_Status;
		Pin17FB: FB_Cylinder_Status;
		Pin18FB: FB_Cylinder_Status;
		Slide1FB: FB_Cylinder_Status;
		Slide2FB: FB_Cylinder_Status;
		Slide3FB: FB_Cylinder_Status;
		Slide4FB: FB_Cylinder_Status;
		Slide5FB: FB_Cylinder_Status;
		Slide6FB: FB_Cylinder_Status;
		Slide7FB: FB_Cylinder_Status;
		Slide8FB: FB_Cylinder_Status;
		Slide9FB: FB_Cylinder_Status;
		Slide10FB: FB_Cylinder_Status;
		Slide11FB: FB_Cylinder_Status;
		Slide12FB: FB_Cylinder_Status;
		Slide13FB: FB_Cylinder_Status;
		Slide14FB: FB_Cylinder_Status;
		Slide15FB: FB_Cylinder_Status;
		Slide16FB: FB_Cylinder_Status;
		Swing1FB: FB_Cylinder_Status;
		Swing2FB: FB_Cylinder_Status;
		Swing3FB: FB_Cylinder_Status;
		Swing4FB: FB_Cylinder_Status;
		Swing5FB: FB_Cylinder_Status;
		Swing6FB: FB_Cylinder_Status;
		QACheck1FB: FB_Cylinder_Status;
		QACheck2FB: FB_Cylinder_Status;
		CheckQA1FB: FB_GTAC_QAcheck_20150529;
		Part_Present1FB: FB_PP_Sensor;
		Part_Present2FB: FB_PP_Sensor;
		Part_Present3FB: FB_PP_Sensor;
		Part_Present4FB: FB_PP_Sensor;
		Part_Present5FB: FB_PP_Sensor;
		Part_Present6FB: FB_PP_Sensor;
		Part_Present7FB: FB_PP_Sensor;
		Part_Present8FB: FB_PP_Sensor;
		Part_Present9FB: FB_PP_Sensor;
		Part_Present10FB: FB_PP_Sensor;
		Part_Present11FB: FB_PP_Sensor;
		Part_Present12FB: FB_PP_Sensor;
		Part_Present13FB: FB_PP_Sensor;
		Part_Present14FB: FB_PP_Sensor;
		Part_Present15FB: FB_PP_Sensor;
		Part_Present16FB: FB_PP_Sensor;
		Part_Present17FB: FB_PP_Sensor;
		Part_Present18FB: FB_PP_Sensor;
		Part_Present19FB: FB_PP_Sensor;
		Part_Present20FB: FB_PP_Sensor;
		Part_Present21FB: FB_PP_Sensor;
		Part_Present22FB: FB_PP_Sensor;
		Part_Present23FB: FB_PP_Sensor;
		Part_Present24FB: FB_PP_Sensor;
		Part_Present25FB: FB_PP_Sensor;
		Part_Present26FB: FB_PP_Sensor;
		Part_Present27FB: FB_PP_Sensor;
		Part_Present28FB: FB_PP_Sensor;
		Part_Present29FB: FB_PP_Sensor;
		Part_Present30FB: FB_PP_Sensor;
		Part_Present31FB: FB_PP_Sensor;
		Part_Present32FB: FB_PP_Sensor;
		Part_Present33FB: FB_PP_Sensor;
		Part_Present34FB: FB_PP_Sensor;
		Part_Present35FB: FB_PP_Sensor;
		Part_Present36FB: FB_PP_Sensor;
		Part_Present37FB: FB_PP_Sensor;
		Part_Present38FB: FB_PP_Sensor;
		Part_Present39FB: FB_PP_Sensor;
		Part_Present40FB: FB_PP_Sensor;
		Tape_Present1FB: FB_PP_Sensor;

		(*Valve FBs*)
		Valve1FB: FB_GTAC_Valve_20170704;
		Valve2FB: FB_GTAC_Valve_20170704;
		Valve3FB: FB_GTAC_Valve_20170704;
		Valve4FB: FB_GTAC_Valve_20170704;
		Valve5FB: FB_GTAC_Valve_20170704;
		Valve6FB: FB_GTAC_Valve_20170704;
		Valve7FB: FB_GTAC_Valve_20170704;
		Valve8FB: FB_GTAC_Valve_20170704;
		Valve9FB: FB_GTAC_Valve_20170704;
		Valve10FB: FB_GTAC_Valve_20170704;
		Valve11FB: FB_GTAC_Valve_20170704;
		Valve12FB: FB_GTAC_Valve_20170704;
		Valve13FB: FB_GTAC_Valve_20170704;
		Valve14FB: FB_GTAC_Valve_20170704;
		Valve15FB: FB_GTAC_Valve_20170704;
		Valve16FB: FB_GTAC_Valve_20170704;
		Valve17FB: FB_GTAC_Valve_20170704;
		Valve18FB: FB_GTAC_Valve_20170704;
		Valve19FB: FB_GTAC_Valve_20170704;
		Valve20FB: FB_GTAC_Valve_20170704;
		Valve21FB: FB_GTAC_Valve_20170704;
		Valve22FB: FB_GTAC_Valve_20170704;
		Valve23FB: FB_GTAC_Valve_20170704;
		Valve24FB: FB_GTAC_Valve_20170704;
		Valve25FB: FB_GTAC_Valve_20170704;
		Valve26FB: FB_GTAC_Valve_20170704;
		Valve27FB: FB_GTAC_Valve_20170704;
		Valve28FB: FB_GTAC_Valve_20170704;
		Valve29FB: FB_GTAC_Valve_20170704;
		Valve30FB: FB_GTAC_Valve_20170704;
		Valve31FB: FB_GTAC_Valve_20170704;
		Valve32FB: FB_GTAC_Valve_20170704;
		Valve33FB: FB_GTAC_Valve_20170704;
		Valve34FB: FB_GTAC_Valve_20170704;
		Valve35FB: FB_GTAC_Valve_20170704;
		Valve36FB: FB_GTAC_Valve_20170704;
		Valve37FB: FB_GTAC_Valve_20170704;
		Valve38FB: FB_GTAC_Valve_20170704;
		Valve39FB: FB_GTAC_Valve_20170704;
		Valve40FB: FB_GTAC_Valve_20170704;
		Valve41FB: FB_GTAC_Valve_20170704;
		Valve42FB: FB_GTAC_Valve_20170704;
		Valve43FB: FB_GTAC_Valve_20170704;
		Valve44FB: FB_GTAC_Valve_20170704;
		Valve45FB: FB_GTAC_Valve_20170704;
		Valve46FB: FB_GTAC_Valve_20170704;
		Valve47FB: FB_GTAC_Valve_20170704;
		Valve48FB: FB_GTAC_Valve_20170704;

		(*Tool Positions*)
			(*Add User Indivdual Position Variables Here*)
			Clamp1ADVD: BOOL;
			Clamp1RETD: BOOL;
			Clamp2ADVD: BOOL;
			Clamp2RETD: BOOL;
			Clamp3ADVD: BOOL;
			Clamp3RETD: BOOL;
			Clamp4ADVD: BOOL;
			Clamp4RETD: BOOL;
			Clamp5ADVD: BOOL;
			Clamp5RETD: BOOL;
			Clamp6ADVD: BOOL;
			Clamp6RETD: BOOL;
			Clamp7ADVD: BOOL;
			Clamp7RETD: BOOL;
			Clamp8ADVD: BOOL;
			Clamp8RETD: BOOL;
			Clamp9ADVD: BOOL;
			Clamp9RETD: BOOL;
			Clamp10ADVD: BOOL;
			Clamp10RETD: BOOL;
			Clamp11ADVD: BOOL;
			Clamp11RETD: BOOL;
			Clamp12ADVD: BOOL;
			Clamp12RETD: BOOL;
			Clamp13ADVD: BOOL;
			Clamp13RETD: BOOL;
			Clamp14ADVD: BOOL;
			Clamp14RETD: BOOL;
			Clamp15ADVD: BOOL;
			Clamp15RETD: BOOL;
			Clamp16ADVD: BOOL;
			Clamp16RETD: BOOL;
			Clamp17ADVD: BOOL;
			Clamp17RETD: BOOL;
			Clamp18ADVD: BOOL;
			Clamp18RETD: BOOL;
			Clamp19ADVD: BOOL;
			Clamp19RETD: BOOL;
			Clamp20ADVD: BOOL;
			Clamp20RETD: BOOL;
			Clamp21ADVD: BOOL;
			Clamp21RETD: BOOL;
			Clamp22ADVD: BOOL;
			Clamp22RETD: BOOL;
			Clamp23ADVD: BOOL;
			Clamp23RETD: BOOL;
			Clamp24ADVD: BOOL;
			Clamp24RETD: BOOL;
			Cyl1ADVD: BOOL;
			Cyl1MID: BOOL;
			Cyl1RETD: BOOL;
			Pin1ADVD: BOOL;
			Pin1RETD: BOOL;
			Pin2ADVD: BOOL;
			Pin2RETD: BOOL;
			Pin3ADVD: BOOL;
			Pin3RETD: BOOL;
			Pin4ADVD: BOOL;
			Pin4RETD: BOOL;
			Pin5ADVD: BOOL;
			Pin5RETD: BOOL;
			Pin6ADVD: BOOL;
			Pin6RETD: BOOL;
			Pin7ADVD: BOOL;
			Pin7RETD: BOOL;
			Pin8ADVD: BOOL;
			Pin8RETD: BOOL;
			Pin9ADVD: BOOL;
			Pin9RETD: BOOL;
			Pin10ADVD: BOOL;
			Pin10RETD: BOOL;
			Pin11ADVD: BOOL;
			Pin11RETD: BOOL;
			Pin12ADVD: BOOL;
			Pin12RETD: BOOL;
			Pin13ADVD: BOOL;
			Pin13RETD: BOOL;
			Pin14ADVD: BOOL;
			Pin14RETD: BOOL;
			Pin15ADVD: BOOL;
			Pin15RETD: BOOL;
			Pin16ADVD: BOOL;
			Pin16RETD: BOOL;
			Pin17ADVD: BOOL;
			Pin17RETD: BOOL;
			Pin18ADVD: BOOL;
			Pin18RETD: BOOL;
			Slide1ADVD: BOOL;
			Slide1RETD: BOOL;
			Slide2ADVD: BOOL;
			Slide2RETD: BOOL;
			Slide3ADVD: BOOL;
			Slide3RETD: BOOL;
			Slide4ADVD: BOOL;
			Slide4RETD: BOOL;
			Slide5ADVD: BOOL;
			Slide5RETD: BOOL;
			Slide6ADVD: BOOL;
			Slide6RETD: BOOL;
			Slide7ADVD: BOOL;
			Slide7RETD: BOOL;
			Slide8ADVD: BOOL;
			Slide8RETD: BOOL;
			Slide9ADVD: BOOL;
			Slide9RETD: BOOL;
			Slide10ADVD: BOOL;
			Slide10RETD: BOOL;
			Slide11ADVD: BOOL;
			Slide11RETD: BOOL;
			Slide12ADVD: BOOL;
			Slide12RETD: BOOL;
			Slide13ADVD: BOOL;
			Slide13RETD: BOOL;
			Slide14ADVD: BOOL;
			Slide14RETD: BOOL;
			Slide15ADVD: BOOL;
			Slide15RETD: BOOL;
			Slide16ADVD: BOOL;
			Slide16RETD: BOOL;
			Swing1ADVD: BOOL;
			Swing1RETD: BOOL;
			Swing2ADVD: BOOL;
			Swing2RETD: BOOL;
			Swing3ADVD: BOOL;
			Swing3RETD: BOOL;
			Swing4ADVD: BOOL;
			Swing4RETD: BOOL;
			Swing5ADVD: BOOL;
			Swing5RETD: BOOL;
			Swing6ADVD: BOOL;
			Swing6RETD: BOOL;
			QACheck1ADVD: BOOL;
			QACheck1RETD: BOOL;
			QACheck2ADVD: BOOL;
			QACheck2RETD: BOOL;

